nErrorCode := fbMlSvr.nErrorCode;
nMaxInferenceDuration := fbMlSvr.nMaxInferenceDuration;

END_FUNCTION_BLOCK

// ---- POUs/FB_PeriodicLstmSequenceTf3820Runner.TcPOU
FUNCTION_BLOCK FB_PeriodicLstmSequenceTf3820Runner
VAR_INPUT
	sModelJsonFilePath	: T_MaxString;
	sMlSvrNetId			: T_MaxString := 'local';
	eExecutionProvider	: E_ExecutionProvider := E_ExecutionProvider.CPU;
	bEnable				: BOOL;
	bReset					: BOOL;
	bLoadModel			: BOOL;
	nConfigureTimeout	: UDINT := 1000;
	nPredictTimeout		: UDINT := 100;
	nPriority			: UDINT := 0;
	fTheta					: REAL;
	fThetaDot				: REAL;
	fTorque				: REAL;
	fTemperature			: REAL;
	fDirectionFlag		: REAL;
	fThetaStep			: REAL := 0.25;
END_VAR
VAR
	fbMlSvr				: FB_MlSvrPrediction;
	stModelInput		: ST_PeriodicLstmSequenceInput;
	stModelOutput		: ST_PeriodicLstmSequenceOutput;
	rtrig_model			: R_TRIG;
	nState					: INT := 0;
	nSequenceIndex		: INT;
	nOutputIndex		: INT;
END_VAR
VAR_OUTPUT
	bConfigured			: BOOL;
	bBusy					: BOOL;
	bPredictionPending	: BOOL;
	bPredictionReady	: BOOL;
	bResetDone			: BOOL;
	bError					: BOOL;
	nErrorCode			: HRESULT;
	nMaxInferenceDuration	: UDINT;
	aPredictionOutput	: ARRAY[0..8] OF REAL;
END_VAR

rtrig_model(CLK := bLoadModel);

IF rtrig_model.Q THEN
	bPredictionPending := FALSE;
	bPredictionReady := FALSE;
	bResetDone := FALSE;
	bError := FALSE;
	IF fbMlSvr.bConfigured THEN
		nState := 5;
	ELSE
		bConfigured := FALSE;
		nState := 10;
	END_IF
END_IF

IF bReset THEN
	bPredictionPending := FALSE;
	bPredictionReady := FALSE;
	bError := FALSE;
	IF fbMlSvr.bConfigured THEN
		nState := 5;
	ELSE
		bConfigured := FALSE;
		bResetDone := TRUE;
		nState := 0;
	END_IF
END_IF

CASE nState OF
	0:
		bBusy := FALSE;
		IF bLoadModel AND NOT(bConfigured) AND NOT(bReset) THEN
			nState := 10;
		END_IF

	5:
		bBusy := TRUE;
		IF fbMlSvr.Deconfigure(nTimeout := nConfigureTimeout) THEN
			nErrorCode := fbMlSvr.nErrorCode;
			bError := fbMlSvr.bError OR (nErrorCode <> 0);
			bConfigured := FALSE;
			bBusy := FALSE;
			bResetDone := NOT(bError);
			IF bError THEN
				nState := 90;
			ELSIF bReset THEN
				nState := 0;
			ELSE
				nState := 10;
			END_IF
		END_IF

	10:
		bBusy := TRUE;
		fbMlSvr.stPredictionParameter.sMlModelFilePath := sModelJsonFilePath;
		fbMlSvr.stPredictionParameter.sMlSvrNetId := sMlSvrNetId;
		fbMlSvr.stPredictionParameter.eExecutionProvider := eExecutionProvider;
		IF fbMlSvr.Configure(nTimeout := nConfigureTimeout, nPriority := nPriority) THEN
			nErrorCode := fbMlSvr.nErrorCode;
			bError := fbMlSvr.bError OR (nErrorCode <> 0);
			bConfigured := fbMlSvr.bConfigured AND NOT(bError);
			bBusy := FALSE;
			IF bConfigured THEN
				nState := 20;
			ELSE
				nState := 90;
			END_IF
		END_IF

	20:
		bBusy := FALSE;
		bPredictionPending := FALSE;
		IF bEnable AND bConfigured AND NOT(bError) AND NOT(bReset) THEN
			FOR nSequenceIndex := 0 TO 32 DO
				stModelInput.in_input_tensor[0,nSequenceIndex,0] := fTheta + (INT_TO_REAL(nSequenceIndex) * fThetaStep);
				stModelInput.in_input_tensor[0,nSequenceIndex,1] := fThetaDot;
				stModelInput.in_input_tensor[0,nSequenceIndex,2] := fTorque;
				stModelInput.in_input_tensor[0,nSequenceIndex,3] := fTemperature;
				stModelInput.in_input_tensor[0,nSequenceIndex,4] := fDirectionFlag;
			END_FOR
			bPredictionReady := FALSE;
			bPredictionPending := TRUE;
			nState := 30;
		END_IF

	30:
		bBusy := TRUE;
		bPredictionPending := TRUE;
		IF fbMlSvr.Predict(
			pDataIn := ADR(stModelInput),
			nDataInSize := SIZEOF(ST_PeriodicLstmSequenceInput),
			pDataOut := ADR(stModelOutput),
			nDataOutSize := SIZEOF(ST_PeriodicLstmSequenceOutput),
			nTimeout := nPredictTimeout,
			nPriority := nPriority) THEN
			nErrorCode := fbMlSvr.nErrorCode;
			bError := fbMlSvr.bError OR (nErrorCode <> 0);
			nMaxInferenceDuration := fbMlSvr.nMaxInferenceDuration;
			bPredictionPending := FALSE;
			bBusy := FALSE;
			IF NOT(bError) THEN
				aPredictionOutput[0] := stModelOutput.out_prediction_tensor[0,0];
				FOR nOutputIndex := 1 TO 8 DO
					aPredictionOutput[nOutputIndex] := 0.0;
				END_FOR
				bPredictionReady := TRUE;
				nState := 20;
			ELSE
				nState := 90;
			END_IF
		END_IF

	90:
		bBusy := FALSE;
		bPredictionPending := FALSE;
		bError := TRUE;
END_CASE

nErrorCode := fbMlSvr.nErrorCode;
nMaxInferenceDuration := fbMlSvr.nMaxInferenceDuration;

END_FUNCTION_BLOCK

// ---- POUs/FB_PeriodicMlpTf3820Runner.TcPOU
FUNCTION_BLOCK FB_PeriodicMlpTf3820Runner
VAR_INPUT
	sModelJsonFilePath	: T_MaxString;
	sMlSvrNetId			: T_MaxString := 'local';
	eExecutionProvider	: E_ExecutionProvider := E_ExecutionProvider.CPU;
	bEnable				: BOOL;
	bReset					: BOOL;
	bLoadModel			: BOOL;
	nConfigureTimeout	: UDINT := 1000;
	nPredictTimeout		: UDINT := 100;
	nPriority			: UDINT := 0;
	fTheta					: REAL;
	fThetaDot				: REAL;
	fTorque				: REAL;
	fTemperature			: REAL;
	fDirectionFlag		: REAL;
	fThetaStep			: REAL := 0.25;
END_VAR
VAR
	fbMlSvr				: FB_MlSvrPrediction;
	stModelInput		: ST_PeriodicMlpInput;
	stModelOutput		: ST_PeriodicMlpOutput;
	rtrig_model			: R_TRIG;
	nState					: INT := 0;
	nSequenceIndex		: INT;
	nOutputIndex		: INT;
END_VAR
VAR_OUTPUT
	bConfigured			: BOOL;
	bBusy					: BOOL;
	bPredictionPending	: BOOL;
	bPredictionReady	: BOOL;
	bResetDone			: BOOL;
	bError					: BOOL;
	nErrorCode			: HRESULT;
	nMaxInferenceDuration	: UDINT;
	aPredictionOutput	: ARRAY[0..8] OF REAL;
END_VAR

rtrig_model(CLK := bLoadModel);

IF rtrig_model.Q THEN
	bPredictionPending := FALSE;
	bPredictionReady := FALSE;
	bResetDone := FALSE;
	bError := FALSE;
	IF fbMlSvr.bConfigured THEN
		nState := 5;
	ELSE
		bConfigured := FALSE;
		nState := 10;
	END_IF
END_IF

IF bReset THEN
	bPredictionPending := FALSE;
	bPredictionReady := FALSE;
	bError := FALSE;
	IF fbMlSvr.bConfigured THEN
		nState := 5;
	ELSE
		bConfigured := FALSE;
		bResetDone := TRUE;
		nState := 0;
	END_IF
END_IF

CASE nState OF
	0:
		bBusy := FALSE;
		IF bLoadModel AND NOT(bConfigured) AND NOT(bReset) THEN
			nState := 10;
		END_IF

	5:
		bBusy := TRUE;
		IF fbMlSvr.Deconfigure(nTimeout := nConfigureTimeout) THEN
			nErrorCode := fbMlSvr.nErrorCode;
			bError := fbMlSvr.bError OR (nErrorCode <> 0);
			bConfigured := FALSE;
			bBusy := FALSE;
			bResetDone := NOT(bError);
			IF bError THEN
				nState := 90;
			ELSIF bReset THEN
				nState := 0;
			ELSE
				nState := 10;
			END_IF
		END_IF

	10:
		bBusy := TRUE;
		fbMlSvr.stPredictionParameter.sMlModelFilePath := sModelJsonFilePath;
		fbMlSvr.stPredictionParameter.sMlSvrNetId := sMlSvrNetId;
		fbMlSvr.stPredictionParameter.eExecutionProvider := eExecutionProvider;
		IF fbMlSvr.Configure(nTimeout := nConfigureTimeout, nPriority := nPriority) THEN
			nErrorCode := fbMlSvr.nErrorCode;
			bError := fbMlSvr.bError OR (nErrorCode <> 0);
			bConfigured := fbMlSvr.bConfigured AND NOT(bError);
			bBusy := FALSE;
			IF bConfigured THEN
				nState := 20;
			ELSE
				nState := 90;
			END_IF
		END_IF

	20:
		bBusy := FALSE;
		bPredictionPending := FALSE;
		IF bEnable AND bConfigured AND NOT(bError) AND NOT(bReset) THEN
			stModelInput.in_input_tensor[0,0] := fTheta;
			stModelInput.in_input_tensor[0,1] := fThetaDot;
			stModelInput.in_input_tensor[0,2] := fTorque;
			stModelInput.in_input_tensor[0,3] := fTemperature;
			stModelInput.in_input_tensor[0,4] := fDirectionFlag;
			bPredictionReady := FALSE;
			bPredictionPending := TRUE;
			nState := 30;
		END_IF

	30:
		bBusy := TRUE;
		bPredictionPending := TRUE;
		IF fbMlSvr.Predict(
			pDataIn := ADR(stModelInput),
			nDataInSize := SIZEOF(ST_PeriodicMlpInput),
			pDataOut := ADR(stModelOutput),
			nDataOutSize := SIZEOF(ST_PeriodicMlpOutput),
			nTimeout := nPredictTimeout,
			nPriority := nPriority) THEN
			nErrorCode := fbMlSvr.nErrorCode;
			bError := fbMlSvr.bError OR (nErrorCode <> 0);
			nMaxInferenceDuration := fbMlSvr.nMaxInferenceDuration;
			bPredictionPending := FALSE;
			bBusy := FALSE;
			IF NOT(bError) THEN
				aPredictionOutput[0] := stModelOutput.out_prediction_tensor[0,0];
				FOR nOutputIndex := 1 TO 8 DO
					aPredictionOutput[nOutputIndex] := 0.0;
				END_FOR
				bPredictionReady := TRUE;
				nState := 20;
			ELSE
				nState := 90;
			END_IF
		END_IF

	90:
		bBusy := FALSE;
		bPredictionPending := FALSE;
		bError := TRUE;
END_CASE

nErrorCode := fbMlSvr.nErrorCode;
nMaxInferenceDuration := fbMlSvr.nMaxInferenceDuration;

END_FUNCTION_BLOCK

// ---- POUs/FB_PeriodicMlpHarmonicTf3820Runner.TcPOU
FUNCTION_BLOCK FB_PeriodicMlpHarmonicTf3820Runner
VAR_INPUT
	sModelJsonFilePath	: T_MaxString;
	sMlSvrNetId			: T_MaxString := 'local';
	eExecutionProvider	: E_ExecutionProvider := E_ExecutionProvider.CPU;
	bEnable				: BOOL;
	bReset					: BOOL;
	bLoadModel			: BOOL;
	nConfigureTimeout	: UDINT := 1000;
	nPredictTimeout		: UDINT := 100;
	nPriority			: UDINT := 0;
	fTheta					: REAL;
	fThetaDot				: REAL;
	fTorque				: REAL;
	fTemperature			: REAL;
	fDirectionFlag		: REAL;
	fThetaStep			: REAL := 0.25;
END_VAR
VAR
	fbMlSvr				: FB_MlSvrPrediction;
	stModelInput		: ST_PeriodicMlpHarmonicInput;
	stModelOutput		: ST_PeriodicMlpHarmonicOutput;
	rtrig_model			: R_TRIG;
	nState					: INT := 0;
	nSequenceIndex		: INT;
	nOutputIndex		: INT;
END_VAR
VAR_OUTPUT
	bConfigured			: BOOL;
	bBusy					: BOOL;
	bPredictionPending	: BOOL;
	bPredictionReady	: BOOL;
	bResetDone			: BOOL;
	bError					: BOOL;
	nErrorCode			: HRESULT;
	nMaxInferenceDuration	: UDINT;
	aPredictionOutput	: ARRAY[0..8] OF REAL;
END_VAR

rtrig_model(CLK := bLoadModel);

IF rtrig_model.Q THEN
	bPredictionPending := FALSE;
	bPredictionReady := FALSE;
	bResetDone := FALSE;
	bError := FALSE;
	IF fbMlSvr.bConfigured THEN
		nState := 5;
	ELSE
		bConfigured := FALSE;
		nState := 10;
	END_IF
END_IF

IF bReset THEN
	bPredictionPending := FALSE;
	bPredictionReady := FALSE;
	bError := FALSE;
	IF fbMlSvr.bConfigured THEN
		nState := 5;
	ELSE
		bConfigured := FALSE;
		bResetDone := TRUE;
		nState := 0;
	END_IF
END_IF

CASE nState OF
	0:
		bBusy := FALSE;
		IF bLoadModel AND NOT(bConfigured) AND NOT(bReset) THEN
			nState := 10;
		END_IF

	5:
		bBusy := TRUE;
		IF fbMlSvr.Deconfigure(nTimeout := nConfigureTimeout) THEN
			nErrorCode := fbMlSvr.nErrorCode;
			bError := fbMlSvr.bError OR (nErrorCode <> 0);
			bConfigured := FALSE;
			bBusy := FALSE;
			bResetDone := NOT(bError);
			IF bError THEN
				nState := 90;
			ELSIF bReset THEN
				nState := 0;
			ELSE
				nState := 10;
			END_IF
		END_IF

	10:
		bBusy := TRUE;
		fbMlSvr.stPredictionParameter.sMlModelFilePath := sModelJsonFilePath;
		fbMlSvr.stPredictionParameter.sMlSvrNetId := sMlSvrNetId;
		fbMlSvr.stPredictionParameter.eExecutionProvider := eExecutionProvider;
		IF fbMlSvr.Configure(nTimeout := nConfigureTimeout, nPriority := nPriority) THEN
			nErrorCode := fbMlSvr.nErrorCode;
			bError := fbMlSvr.bError OR (nErrorCode <> 0);
			bConfigured := fbMlSvr.bConfigured AND NOT(bError);
			bBusy := FALSE;
			IF bConfigured THEN
				nState := 20;
			ELSE
				nState := 90;
			END_IF
		END_IF

	20:
		bBusy := FALSE;
		bPredictionPending := FALSE;
		IF bEnable AND bConfigured AND NOT(bError) AND NOT(bReset) THEN
			stModelInput.in_input_tensor[0,0] := fTheta;
			stModelInput.in_input_tensor[0,1] := fThetaDot;
			stModelInput.in_input_tensor[0,2] := fTorque;
			stModelInput.in_input_tensor[0,3] := fTemperature;
			stModelInput.in_input_tensor[0,4] := fDirectionFlag;
			bPredictionReady := FALSE;
			bPredictionPending := TRUE;
			nState := 30;
		END_IF

	30:
		bBusy := TRUE;
		bPredictionPending := TRUE;
		IF fbMlSvr.Predict(
			pDataIn := ADR(stModelInput),
			nDataInSize := SIZEOF(ST_PeriodicMlpHarmonicInput),
			pDataOut := ADR(stModelOutput),
			nDataOutSize := SIZEOF(ST_PeriodicMlpHarmonicOutput),
			nTimeout := nPredictTimeout,
			nPriority := nPriority) THEN
			nErrorCode := fbMlSvr.nErrorCode;
			bError := fbMlSvr.bError OR (nErrorCode <> 0);
			nMaxInferenceDuration := fbMlSvr.nMaxInferenceDuration;
			bPredictionPending := FALSE;
			bBusy := FALSE;
			IF NOT(bError) THEN
				aPredictionOutput[0] := stModelOutput.out_prediction_tensor[0,0];
				FOR nOutputIndex := 1 TO 8 DO
					aPredictionOutput[nOutputIndex] := 0.0;
				END_FOR
				bPredictionReady := TRUE;
				nState := 20;
			ELSE
				nState := 90;
			END_IF
		END_IF

	90:
		bBusy := FALSE;
		bPredictionPending := FALSE;
		bError := TRUE;
END_CASE

nErrorCode := fbMlSvr.nErrorCode;
nMaxInferenceDuration := fbMlSvr.nMaxInferenceDuration;

END_FUNCTION_BLOCK

// ---- POUs/FB_PeriodicTemporalConvolutionTf3820Runner.TcPOU
FUNCTION_BLOCK FB_PeriodicTemporalConvolutionTf3820Runner
VAR_INPUT
	sModelJsonFilePath	: T_MaxString;
	sMlSvrNetId			: T_MaxString := 'local';
	eExecutionProvider	: E_ExecutionProvider := E_ExecutionProvider.CPU;
	bEnable				: BOOL;
	bReset					: BOOL;
	bLoadModel			: BOOL;
	nConfigureTimeout	: UDINT := 1000;
	nPredictTimeout		: UDINT := 100;
	nPriority			: UDINT := 0;
	fTheta					: REAL;
	fThetaDot				: REAL;
	fTorque				: REAL;
	fTemperature			: REAL;
	fDirectionFlag		: REAL;
	fThetaStep			: REAL := 0.25;
END_VAR
VAR
	fbMlSvr				: FB_MlSvrPrediction;
	stModelInput		: ST_PeriodicTemporalConvolutionInput;
	stModelOutput		: ST_PeriodicTemporalConvolutionOutput;
	rtrig_model			: R_TRIG;
	nState					: INT := 0;
	nSequenceIndex		: INT;
	nOutputIndex		: INT;
END_VAR
VAR_OUTPUT
	bConfigured			: BOOL;
	bBusy					: BOOL;
	bPredictionPending	: BOOL;
	bPredictionReady	: BOOL;
	bResetDone			: BOOL;
	bError					: BOOL;
	nErrorCode			: HRESULT;
	nMaxInferenceDuration	: UDINT;
	aPredictionOutput	: ARRAY[0..8] OF REAL;
END_VAR

rtrig_model(CLK := bLoadModel);

IF rtrig_model.Q THEN
	bPredictionPending := FALSE;
	bPredictionReady := FALSE;
	bResetDone := FALSE;
	bError := FALSE;
	IF fbMlSvr.bConfigured THEN
		nState := 5;
	ELSE
		bConfigured := FALSE;
		nState := 10;
	END_IF
END_IF

IF bReset THEN
	bPredictionPending := FALSE;
	bPredictionReady := FALSE;
	bError := FALSE;
	IF fbMlSvr.bConfigured THEN
		nState := 5;
	ELSE
		bConfigured := FALSE;
		bResetDone := TRUE;
		nState := 0;
	END_IF
END_IF

CASE nState OF
	0:
		bBusy := FALSE;
		IF bLoadModel AND NOT(bConfigured) AND NOT(bReset) THEN
			nState := 10;
		END_IF

	5:
		bBusy := TRUE;
		IF fbMlSvr.Deconfigure(nTimeout := nConfigureTimeout) THEN
			nErrorCode := fbMlSvr.nErrorCode;
			bError := fbMlSvr.bError OR (nErrorCode <> 0);
			bConfigured := FALSE;
			bBusy := FALSE;
			bResetDone := NOT(bError);
			IF bError THEN
				nState := 90;
			ELSIF bReset THEN
				nState := 0;
			ELSE
				nState := 10;
			END_IF
		END_IF

	10:
		bBusy := TRUE;
		fbMlSvr.stPredictionParameter.sMlModelFilePath := sModelJsonFilePath;
		fbMlSvr.stPredictionParameter.sMlSvrNetId := sMlSvrNetId;
		fbMlSvr.stPredictionParameter.eExecutionProvider := eExecutionProvider;
		IF fbMlSvr.Configure(nTimeout := nConfigureTimeout, nPriority := nPriority) THEN
			nErrorCode := fbMlSvr.nErrorCode;
			bError := fbMlSvr.bError OR (nErrorCode <> 0);
			bConfigured := fbMlSvr.bConfigured AND NOT(bError);
			bBusy := FALSE;
			IF bConfigured THEN
				nState := 20;
			ELSE
				nState := 90;
			END_IF
		END_IF

	20:
		bBusy := FALSE;
		bPredictionPending := FALSE;
		IF bEnable AND bConfigured AND NOT(bError) AND NOT(bReset) THEN
			FOR nSequenceIndex := 0 TO 32 DO
				stModelInput.in_input_tensor[0,nSequenceIndex,0] := fTheta + (INT_TO_REAL(nSequenceIndex) * fThetaStep);
				stModelInput.in_input_tensor[0,nSequenceIndex,1] := fThetaDot;
				stModelInput.in_input_tensor[0,nSequenceIndex,2] := fTorque;
				stModelInput.in_input_tensor[0,nSequenceIndex,3] := fTemperature;
				stModelInput.in_input_tensor[0,nSequenceIndex,4] := fDirectionFlag;
			END_FOR
			bPredictionReady := FALSE;
			bPredictionPending := TRUE;
			nState := 30;
		END_IF

	30:
		bBusy := TRUE;
		bPredictionPending := TRUE;
		IF fbMlSvr.Predict(
			pDataIn := ADR(stModelInput),
			nDataInSize := SIZEOF(ST_PeriodicTemporalConvolutionInput),
			pDataOut := ADR(stModelOutput),
			nDataOutSize := SIZEOF(ST_PeriodicTemporalConvolutionOutput),
			nTimeout := nPredictTimeout,
			nPriority := nPriority) THEN
			nErrorCode := fbMlSvr.nErrorCode;
			bError := fbMlSvr.bError OR (nErrorCode <> 0);
			nMaxInferenceDuration := fbMlSvr.nMaxInferenceDuration;
			bPredictionPending := FALSE;
			bBusy := FALSE;
			IF NOT(bError) THEN
				aPredictionOutput[0] := stModelOutput.out_prediction_tensor[0,0];
				FOR nOutputIndex := 1 TO 8 DO
					aPredictionOutput[nOutputIndex] := 0.0;
				END_FOR
				bPredictionReady := TRUE;
				nState := 20;
			ELSE
				nState := 90;
			END_IF
		END_IF

	90:
		bBusy := FALSE;
		bPredictionPending := FALSE;
		bError := TRUE;
END_CASE

nErrorCode := fbMlSvr.nErrorCode;
nMaxInferenceDuration := fbMlSvr.nMaxInferenceDuration;

END_FUNCTION_BLOCK

// ---- POUs/FB_RcimTrack1Tf3820Runner.TcPOU
FUNCTION_BLOCK FB_RcimTrack1Tf3820Runner
VAR_INPUT
	sModelJsonFilePath	: T_MaxString;
	sMlSvrNetId			: T_MaxString := 'local';
	eExecutionProvider	: E_ExecutionProvider := E_ExecutionProvider.CPU;
	bEnable				: BOOL;
	bReset					: BOOL;
	bLoadModel			: BOOL;
	nConfigureTimeout	: UDINT := 1000;
	nPredictTimeout		: UDINT := 100;
	nPriority			: UDINT := 0;
	fTheta					: REAL;
	fThetaDot				: REAL;
	fTorque				: REAL;
	fTemperature			: REAL;
	fDirectionFlag		: REAL;
	fThetaStep			: REAL := 0.25;
END_VAR
VAR
	fbMlSvr				: FB_MlSvrPrediction;
	stModelInput		: ST_RcimTrack1Input;
	stModelOutput		: ST_RcimTrack1Output;
	rtrig_model			: R_TRIG;
	nState					: INT := 0;
	nSequenceIndex		: INT;
	nOutputIndex		: INT;
END_VAR
VAR_OUTPUT
	bConfigured			: BOOL;
	bBusy					: BOOL;
	bPredictionPending	: BOOL;
	bPredictionReady	: BOOL;
	bResetDone			: BOOL;
	bError					: BOOL;
	nErrorCode			: HRESULT;
	nMaxInferenceDuration	: UDINT;
	aPredictionOutput	: ARRAY[0..8] OF REAL;
END_VAR

rtrig_model(CLK := bLoadModel);

IF rtrig_model.Q THEN
	bPredictionPending := FALSE;
	bPredictionReady := FALSE;
	bResetDone := FALSE;
	bError := FALSE;
	IF fbMlSvr.bConfigured THEN
		nState := 5;
	ELSE
		bConfigured := FALSE;
		nState := 10;
	END_IF
END_IF

IF bReset THEN
	bPredictionPending := FALSE;
	bPredictionReady := FALSE;
	bError := FALSE;
	IF fbMlSvr.bConfigured THEN
		nState := 5;
	ELSE
		bConfigured := FALSE;
		bResetDone := TRUE;
		nState := 0;
	END_IF
END_IF

CASE nState OF
	0:
		bBusy := FALSE;
		IF bLoadModel AND NOT(bConfigured) AND NOT(bReset) THEN
			nState := 10;
		END_IF

	5:
		bBusy := TRUE;
		IF fbMlSvr.Deconfigure(nTimeout := nConfigureTimeout) THEN
			nErrorCode := fbMlSvr.nErrorCode;
			bError := fbMlSvr.bError OR (nErrorCode <> 0);
			bConfigured := FALSE;
			bBusy := FALSE;
			bResetDone := NOT(bError);
			IF bError THEN
				nState := 90;
			ELSIF bReset THEN
				nState := 0;
			ELSE
				nState := 10;
			END_IF
		END_IF

	10:
		bBusy := TRUE;
		fbMlSvr.stPredictionParameter.sMlModelFilePath := sModelJsonFilePath;
		fbMlSvr.stPredictionParameter.sMlSvrNetId := sMlSvrNetId;
		fbMlSvr.stPredictionParameter.eExecutionProvider := eExecutionProvider;
		IF fbMlSvr.Configure(nTimeout := nConfigureTimeout, nPriority := nPriority) THEN
			nErrorCode := fbMlSvr.nErrorCode;
			bError := fbMlSvr.bError OR (nErrorCode <> 0);
			bConfigured := fbMlSvr.bConfigured AND NOT(bError);
			bBusy := FALSE;
			IF bConfigured THEN
				nState := 20;
			ELSE
				nState := 90;
			END_IF
		END_IF

	20:
		bBusy := FALSE;
		bPredictionPending := FALSE;
		IF bEnable AND bConfigured AND NOT(bError) AND NOT(bReset) THEN
			stModelInput.in_float_input[0,0] := fThetaDot;
			stModelInput.in_float_input[0,1] := fTemperature;
			stModelInput.in_float_input[0,2] := fTorque;
			bPredictionReady := FALSE;
			bPredictionPending := TRUE;
			nState := 30;
		END_IF

	30:
		bBusy := TRUE;
		bPredictionPending := TRUE;
		IF fbMlSvr.Predict(
			pDataIn := ADR(stModelInput),
			nDataInSize := SIZEOF(ST_RcimTrack1Input),
			pDataOut := ADR(stModelOutput),
			nDataOutSize := SIZEOF(ST_RcimTrack1Output),
			nTimeout := nPredictTimeout,
			nPriority := nPriority) THEN
			nErrorCode := fbMlSvr.nErrorCode;
			bError := fbMlSvr.bError OR (nErrorCode <> 0);
			nMaxInferenceDuration := fbMlSvr.nMaxInferenceDuration;
			bPredictionPending := FALSE;
			bBusy := FALSE;
			IF NOT(bError) THEN
				aPredictionOutput[0] := stModelOutput.out_variable[0,0];
				FOR nOutputIndex := 1 TO 8 DO
					aPredictionOutput[nOutputIndex] := 0.0;
				END_FOR
				bPredictionReady := TRUE;
				nState := 20;
			ELSE
				nState := 90;
			END_IF
		END_IF

	90:
		bBusy := FALSE;
		bPredictionPending := FALSE;
		bError := TRUE;
END_CASE

nErrorCode := fbMlSvr.nErrorCode;
nMaxInferenceDuration := fbMlSvr.nMaxInferenceDuration;

END_FUNCTION_BLOCK

// ---- POUs/FB_ResidualHarmonicGruSequenceDense240Tf3820Runner.TcPOU
FUNCTION_BLOCK FB_ResidualHarmonicGruSequenceDense240Tf3820Runner
VAR_INPUT
	sModelJsonFilePath	: T_MaxString;
	sMlSvrNetId			: T_MaxString := 'local';
	eExecutionProvider	: E_ExecutionProvider := E_ExecutionProvider.CPU;
	bEnable				: BOOL;
	bReset					: BOOL;
	bLoadModel			: BOOL;
	nConfigureTimeout	: UDINT := 1000;
	nPredictTimeout		: UDINT := 100;
	nPriority			: UDINT := 0;
	fTheta					: REAL;
	fThetaDot				: REAL;
	fTorque				: REAL;
	fTemperature			: REAL;
	fDirectionFlag		: REAL;
	fThetaStep			: REAL := 0.25;
END_VAR
VAR
	fbMlSvr				: FB_MlSvrPrediction;
	stModelInput		: ST_ResidualHarmonicGruSequenceDense240Input;
	stModelOutput		: ST_ResidualHarmonicGruSequenceDense240Output;
	rtrig_model			: R_TRIG;
	nState					: INT := 0;
	nSequenceIndex		: INT;
	nOutputIndex		: INT;
END_VAR
VAR_OUTPUT
	bConfigured			: BOOL;
	bBusy					: BOOL;
	bPredictionPending	: BOOL;
	bPredictionReady	: BOOL;
	bResetDone			: BOOL;
	bError					: BOOL;
	nErrorCode			: HRESULT;
	nMaxInferenceDuration	: UDINT;
	aPredictionOutput	: ARRAY[0..8] OF REAL;
END_VAR

rtrig_model(CLK := bLoadModel);

IF rtrig_model.Q THEN
	bPredictionPending := FALSE;
	bPredictionReady := FALSE;
	bResetDone := FALSE;
	bError := FALSE;
	IF fbMlSvr.bConfigured THEN
		nState := 5;
	ELSE
		bConfigured := FALSE;
		nState := 10;
	END_IF
END_IF

IF bReset THEN
	bPredictionPending := FALSE;
	bPredictionReady := FALSE;
	bError := FALSE;
	IF fbMlSvr.bConfigured THEN
		nState := 5;
	ELSE
		bConfigured := FALSE;
		bResetDone := TRUE;
		nState := 0;
	END_IF
END_IF

CASE nState OF
	0:
		bBusy := FALSE;
		IF bLoadModel AND NOT(bConfigured) AND NOT(bReset) THEN
			nState := 10;
		END_IF

	5:
		bBusy := TRUE;
		IF fbMlSvr.Deconfigure(nTimeout := nConfigureTimeout) THEN
			nErrorCode := fbMlSvr.nErrorCode;
			bError := fbMlSvr.bError OR (nErrorCode <> 0);
			bConfigured := FALSE;
			bBusy := FALSE;
			bResetDone := NOT(bError);
			IF bError THEN
				nState := 90;
			ELSIF bReset THEN
				nState := 0;
			ELSE
				nState := 10;
			END_IF
		END_IF

	10:
		bBusy := TRUE;
		fbMlSvr.stPredictionParameter.sMlModelFilePath := sModelJsonFilePath;
		fbMlSvr.stPredictionParameter.sMlSvrNetId := sMlSvrNetId;
		fbMlSvr.stPredictionParameter.eExecutionProvider := eExecutionProvider;
		IF fbMlSvr.Configure(nTimeout := nConfigureTimeout, nPriority := nPriority) THEN
			nErrorCode := fbMlSvr.nErrorCode;
			bError := fbMlSvr.bError OR (nErrorCode <> 0);
			bConfigured := fbMlSvr.bConfigured AND NOT(bError);
			bBusy := FALSE;
			IF bConfigured THEN
				nState := 20;
			ELSE
				nState := 90;
			END_IF
		END_IF

	20:
		bBusy := FALSE;
		bPredictionPending := FALSE;
		IF bEnable AND bConfigured AND NOT(bError) AND NOT(bReset) THEN
			FOR nSequenceIndex := 0 TO 32 DO
				stModelInput.in_input_tensor[0,nSequenceIndex,0] := fTheta + (INT_TO_REAL(nSequenceIndex) * fThetaStep);
				stModelInput.in_input_tensor[0,nSequenceIndex,1] := fThetaDot;
				stModelInput.in_input_tensor[0,nSequenceIndex,2] := fTorque;
				stModelInput.in_input_tensor[0,nSequenceIndex,3] := fTemperature;
				stModelInput.in_input_tensor[0,nSequenceIndex,4] := fDirectionFlag;
			END_FOR
			bPredictionReady := FALSE;
			bPredictionPending := TRUE;
			nState := 30;
		END_IF

	30:
		bBusy := TRUE;
		bPredictionPending := TRUE;
		IF fbMlSvr.Predict(
			pDataIn := ADR(stModelInput),
			nDataInSize := SIZEOF(ST_ResidualHarmonicGruSequenceDense240Input),
			pDataOut := ADR(stModelOutput),
			nDataOutSize := SIZEOF(ST_ResidualHarmonicGruSequenceDense240Output),
			nTimeout := nPredictTimeout,
			nPriority := nPriority) THEN
			nErrorCode := fbMlSvr.nErrorCode;
			bError := fbMlSvr.bError OR (nErrorCode <> 0);
			nMaxInferenceDuration := fbMlSvr.nMaxInferenceDuration;
			bPredictionPending := FALSE;
			bBusy := FALSE;
			IF NOT(bError) THEN
				aPredictionOutput[0] := stModelOutput.out_prediction_tensor[0,0];
				FOR nOutputIndex := 1 TO 8 DO
					aPredictionOutput[nOutputIndex] := 0.0;
				END_FOR
				bPredictionReady := TRUE;
				nState := 20;
			ELSE
				nState := 90;
			END_IF
		END_IF

	90:
		bBusy := FALSE;
		bPredictionPending := FALSE;
		bError := TRUE;
END_CASE

nErrorCode := fbMlSvr.nErrorCode;
nMaxInferenceDuration := fbMlSvr.nMaxInferenceDuration;

END_FUNCTION_BLOCK

// ---- POUs/FB_ResidualHarmonicGruSequenceDense360Tf3820Runner.TcPOU
FUNCTION_BLOCK FB_ResidualHarmonicGruSequenceDense360Tf3820Runner
VAR_INPUT
	sModelJsonFilePath	: T_MaxString;
	sMlSvrNetId			: T_MaxString := 'local';
	eExecutionProvider	: E_ExecutionProvider := E_ExecutionProvider.CPU;
	bEnable				: BOOL;
	bReset					: BOOL;
	bLoadModel			: BOOL;
	nConfigureTimeout	: UDINT := 1000;
	nPredictTimeout		: UDINT := 100;
	nPriority			: UDINT := 0;
	fTheta					: REAL;
	fThetaDot				: REAL;
	fTorque				: REAL;
	fTemperature			: REAL;
	fDirectionFlag		: REAL;
	fThetaStep			: REAL := 0.25;
END_VAR
VAR
	fbMlSvr				: FB_MlSvrPrediction;
	stModelInput		: ST_ResidualHarmonicGruSequenceDense360Input;
	stModelOutput		: ST_ResidualHarmonicGruSequenceDense360Output;
	rtrig_model			: R_TRIG;
	nState					: INT := 0;
	nSequenceIndex		: INT;
	nOutputIndex		: INT;
END_VAR
VAR_OUTPUT
	bConfigured			: BOOL;
	bBusy					: BOOL;
	bPredictionPending	: BOOL;
	bPredictionReady	: BOOL;
	bResetDone			: BOOL;
	bError					: BOOL;
	nErrorCode			: HRESULT;
	nMaxInferenceDuration	: UDINT;
	aPredictionOutput	: ARRAY[0..8] OF REAL;
END_VAR

rtrig_model(CLK := bLoadModel);

IF rtrig_model.Q THEN
	bPredictionPending := FALSE;
	bPredictionReady := FALSE;
	bResetDone := FALSE;
	bError := FALSE;
	IF fbMlSvr.bConfigured THEN
		nState := 5;
	ELSE
		bConfigured := FALSE;
		nState := 10;
	END_IF
END_IF

IF bReset THEN
	bPredictionPending := FALSE;
	bPredictionReady := FALSE;
	bError := FALSE;
	IF fbMlSvr.bConfigured THEN
		nState := 5;
	ELSE
		bConfigured := FALSE;
		bResetDone := TRUE;
		nState := 0;
	END_IF
END_IF

CASE nState OF
	0:
		bBusy := FALSE;
		IF bLoadModel AND NOT(bConfigured) AND NOT(bReset) THEN
			nState := 10;
		END_IF

	5:
		bBusy := TRUE;
		IF fbMlSvr.Deconfigure(nTimeout := nConfigureTimeout) THEN
			nErrorCode := fbMlSvr.nErrorCode;
			bError := fbMlSvr.bError OR (nErrorCode <> 0);
			bConfigured := FALSE;
			bBusy := FALSE;
			bResetDone := NOT(bError);
			IF bError THEN
				nState := 90;
			ELSIF bReset THEN
				nState := 0;
			ELSE
				nState := 10;
			END_IF
		END_IF

	10:
		bBusy := TRUE;
		fbMlSvr.stPredictionParameter.sMlModelFilePath := sModelJsonFilePath;
		fbMlSvr.stPredictionParameter.sMlSvrNetId := sMlSvrNetId;
		fbMlSvr.stPredictionParameter.eExecutionProvider := eExecutionProvider;
		IF fbMlSvr.Configure(nTimeout := nConfigureTimeout, nPriority := nPriority) THEN
			nErrorCode := fbMlSvr.nErrorCode;
			bError := fbMlSvr.bError OR (nErrorCode <> 0);
			bConfigured := fbMlSvr.bConfigured AND NOT(bError);
			bBusy := FALSE;
			IF bConfigured THEN
				nState := 20;
			ELSE
				nState := 90;
			END_IF
		END_IF

	20:
		bBusy := FALSE;
		bPredictionPending := FALSE;
		IF bEnable AND bConfigured AND NOT(bError) AND NOT(bReset) THEN
			FOR nSequenceIndex := 0 TO 32 DO
				stModelInput.in_input_tensor[0,nSequenceIndex,0] := fTheta + (INT_TO_REAL(nSequenceIndex) * fThetaStep);
				stModelInput.in_input_tensor[0,nSequenceIndex,1] := fThetaDot;
				stModelInput.in_input_tensor[0,nSequenceIndex,2] := fTorque;
				stModelInput.in_input_tensor[0,nSequenceIndex,3] := fTemperature;
				stModelInput.in_input_tensor[0,nSequenceIndex,4] := fDirectionFlag;
			END_FOR
			bPredictionReady := FALSE;
			bPredictionPending := TRUE;
			nState := 30;
		END_IF

	30:
		bBusy := TRUE;
		bPredictionPending := TRUE;
		IF fbMlSvr.Predict(
			pDataIn := ADR(stModelInput),
			nDataInSize := SIZEOF(ST_ResidualHarmonicGruSequenceDense360Input),
			pDataOut := ADR(stModelOutput),
			nDataOutSize := SIZEOF(ST_ResidualHarmonicGruSequenceDense360Output),
			nTimeout := nPredictTimeout,
			nPriority := nPriority) THEN
			nErrorCode := fbMlSvr.nErrorCode;
			bError := fbMlSvr.bError OR (nErrorCode <> 0);
			nMaxInferenceDuration := fbMlSvr.nMaxInferenceDuration;
			bPredictionPending := FALSE;
			bBusy := FALSE;
			IF NOT(bError) THEN
				aPredictionOutput[0] := stModelOutput.out_prediction_tensor[0,0];
				FOR nOutputIndex := 1 TO 8 DO
					aPredictionOutput[nOutputIndex] := 0.0;
				END_FOR
				bPredictionReady := TRUE;
				nState := 20;
			ELSE
				nState := 90;
			END_IF
		END_IF

	90:
		bBusy := FALSE;
		bPredictionPending := FALSE;
		bError := TRUE;
END_CASE

nErrorCode := fbMlSvr.nErrorCode;
nMaxInferenceDuration := fbMlSvr.nMaxInferenceDuration;

END_FUNCTION_BLOCK

// ---- POUs/FB_ResidualHarmonicGruSequenceSparseRcimTf3820Runner.TcPOU
FUNCTION_BLOCK FB_ResidualHarmonicGruSequenceSparseRcimTf3820Runner
VAR_INPUT
	sModelJsonFilePath	: T_MaxString;
	sMlSvrNetId			: T_MaxString := 'local';
	eExecutionProvider	: E_ExecutionProvider := E_ExecutionProvider.CPU;
	bEnable				: BOOL;
	bReset					: BOOL;
	bLoadModel			: BOOL;
	nConfigureTimeout	: UDINT := 1000;
	nPredictTimeout		: UDINT := 100;
	nPriority			: UDINT := 0;
	fTheta					: REAL;
	fThetaDot				: REAL;
	fTorque				: REAL;
	fTemperature			: REAL;
	fDirectionFlag		: REAL;
	fThetaStep			: REAL := 0.25;
END_VAR
VAR
	fbMlSvr				: FB_MlSvrPrediction;
	stModelInput		: ST_ResidualHarmonicGruSequenceSparseRcimInput;
	stModelOutput		: ST_ResidualHarmonicGruSequenceSparseRcimOutput;
	rtrig_model			: R_TRIG;
	nState					: INT := 0;
	nSequenceIndex		: INT;
	nOutputIndex		: INT;
END_VAR
VAR_OUTPUT
	bConfigured			: BOOL;
	bBusy					: BOOL;
	bPredictionPending	: BOOL;
	bPredictionReady	: BOOL;
	bResetDone			: BOOL;
	bError					: BOOL;
	nErrorCode			: HRESULT;
	nMaxInferenceDuration	: UDINT;
	aPredictionOutput	: ARRAY[0..8] OF REAL;
END_VAR

rtrig_model(CLK := bLoadModel);

IF rtrig_model.Q THEN
	bPredictionPending := FALSE;
	bPredictionReady := FALSE;
	bResetDone := FALSE;
	bError := FALSE;
	IF fbMlSvr.bConfigured THEN
		nState := 5;
	ELSE
		bConfigured := FALSE;
		nState := 10;
	END_IF
END_IF

IF bReset THEN
	bPredictionPending := FALSE;
	bPredictionReady := FALSE;
	bError := FALSE;
	IF fbMlSvr.bConfigured THEN
		nState := 5;
	ELSE
		bConfigured := FALSE;
		bResetDone := TRUE;
		nState := 0;
	END_IF
END_IF

CASE nState OF
	0:
		bBusy := FALSE;
		IF bLoadModel AND NOT(bConfigured) AND NOT(bReset) THEN
			nState := 10;
		END_IF

	5:
		bBusy := TRUE;
		IF fbMlSvr.Deconfigure(nTimeout := nConfigureTimeout) THEN
			nErrorCode := fbMlSvr.nErrorCode;
			bError := fbMlSvr.bError OR (nErrorCode <> 0);
			bConfigured := FALSE;
			bBusy := FALSE;
			bResetDone := NOT(bError);
			IF bError THEN
				nState := 90;
			ELSIF bReset THEN
				nState := 0;
			ELSE
				nState := 10;
			END_IF
		END_IF

	10:
		bBusy := TRUE;
		fbMlSvr.stPredictionParameter.sMlModelFilePath := sModelJsonFilePath;
		fbMlSvr.stPredictionParameter.sMlSvrNetId := sMlSvrNetId;
		fbMlSvr.stPredictionParameter.eExecutionProvider := eExecutionProvider;
		IF fbMlSvr.Configure(nTimeout := nConfigureTimeout, nPriority := nPriority) THEN
			nErrorCode := fbMlSvr.nErrorCode;
			bError := fbMlSvr.bError OR (nErrorCode <> 0);
			bConfigured := fbMlSvr.bConfigured AND NOT(bError);
			bBusy := FALSE;
			IF bConfigured THEN
				nState := 20;
			ELSE
				nState := 90;
			END_IF
		END_IF

	20:
		bBusy := FALSE;
		bPredictionPending := FALSE;
		IF bEnable AND bConfigured AND NOT(bError) AND NOT(bReset) THEN
			FOR nSequenceIndex := 0 TO 32 DO
				stModelInput.in_input_tensor[0,nSequenceIndex,0] := fTheta + (INT_TO_REAL(nSequenceIndex) * fThetaStep);
				stModelInput.in_input_tensor[0,nSequenceIndex,1] := fThetaDot;
				stModelInput.in_input_tensor[0,nSequenceIndex,2] := fTorque;
				stModelInput.in_input_tensor[0,nSequenceIndex,3] := fTemperature;
				stModelInput.in_input_tensor[0,nSequenceIndex,4] := fDirectionFlag;
			END_FOR
			bPredictionReady := FALSE;
			bPredictionPending := TRUE;
			nState := 30;
		END_IF

	30:
		bBusy := TRUE;
		bPredictionPending := TRUE;
		IF fbMlSvr.Predict(
			pDataIn := ADR(stModelInput),
			nDataInSize := SIZEOF(ST_ResidualHarmonicGruSequenceSparseRcimInput),
			pDataOut := ADR(stModelOutput),
			nDataOutSize := SIZEOF(ST_ResidualHarmonicGruSequenceSparseRcimOutput),
			nTimeout := nPredictTimeout,
			nPriority := nPriority) THEN
			nErrorCode := fbMlSvr.nErrorCode;
			bError := fbMlSvr.bError OR (nErrorCode <> 0);
			nMaxInferenceDuration := fbMlSvr.nMaxInferenceDuration;
			bPredictionPending := FALSE;
			bBusy := FALSE;
			IF NOT(bError) THEN
				aPredictionOutput[0] := stModelOutput.out_prediction_tensor[0,0];
				FOR nOutputIndex := 1 TO 8 DO
					aPredictionOutput[nOutputIndex] := 0.0;
				END_FOR
				bPredictionReady := TRUE;
				nState := 20;
			ELSE
				nState := 90;
			END_IF
		END_IF

	90:
		bBusy := FALSE;
		bPredictionPending := FALSE;
		bError := TRUE;
END_CASE

nErrorCode := fbMlSvr.nErrorCode;
nMaxInferenceDuration := fbMlSvr.nMaxInferenceDuration;

END_FUNCTION_BLOCK

// ---- POUs/FB_ResidualHarmonicLstmSequenceDense240Tf3820Runner.TcPOU
FUNCTION_BLOCK FB_ResidualHarmonicLstmSequenceDense240Tf3820Runner
VAR_INPUT
	sModelJsonFilePath	: T_MaxString;
	sMlSvrNetId			: T_MaxString := 'local';
	eExecutionProvider	: E_ExecutionProvider := E_ExecutionProvider.CPU;
	bEnable				: BOOL;
	bReset					: BOOL;
	bLoadModel			: BOOL;
	nConfigureTimeout	: UDINT := 1000;
	nPredictTimeout		: UDINT := 100;
	nPriority			: UDINT := 0;
	fTheta					: REAL;
	fThetaDot				: REAL;
	fTorque				: REAL;
	fTemperature			: REAL;
	fDirectionFlag		: REAL;
	fThetaStep			: REAL := 0.25;
END_VAR
VAR
	fbMlSvr				: FB_MlSvrPrediction;
	stModelInput		: ST_ResidualHarmonicLstmSequenceDense240Input;
	stModelOutput		: ST_ResidualHarmonicLstmSequenceDense240Output;
	rtrig_model			: R_TRIG;
	nState					: INT := 0;
	nSequenceIndex		: INT;
	nOutputIndex		: INT;
END_VAR
VAR_OUTPUT
	bConfigured			: BOOL;
	bBusy					: BOOL;
	bPredictionPending	: BOOL;
	bPredictionReady	: BOOL;
	bResetDone			: BOOL;
	bError					: BOOL;
	nErrorCode			: HRESULT;
	nMaxInferenceDuration	: UDINT;
	aPredictionOutput	: ARRAY[0..8] OF REAL;
END_VAR

rtrig_model(CLK := bLoadModel);

IF rtrig_model.Q THEN
	bPredictionPending := FALSE;
	bPredictionReady := FALSE;
	bResetDone := FALSE;
	bError := FALSE;
	IF fbMlSvr.bConfigured THEN
		nState := 5;
	ELSE
		bConfigured := FALSE;
		nState := 10;
	END_IF
END_IF

IF bReset THEN
	bPredictionPending := FALSE;
	bPredictionReady := FALSE;
	bError := FALSE;
	IF fbMlSvr.bConfigured THEN
		nState := 5;
	ELSE
		bConfigured := FALSE;
		bResetDone := TRUE;
		nState := 0;
	END_IF
END_IF

CASE nState OF
	0:
		bBusy := FALSE;
		IF bLoadModel AND NOT(bConfigured) AND NOT(bReset) THEN
			nState := 10;
		END_IF

	5:
		bBusy := TRUE;
		IF fbMlSvr.Deconfigure(nTimeout := nConfigureTimeout) THEN
			nErrorCode := fbMlSvr.nErrorCode;
			bError := fbMlSvr.bError OR (nErrorCode <> 0);
			bConfigured := FALSE;
			bBusy := FALSE;
			bResetDone := NOT(bError);
			IF bError THEN
				nState := 90;
			ELSIF bReset THEN
				nState := 0;
			ELSE
				nState := 10;
			END_IF
		END_IF

	10:
		bBusy := TRUE;
		fbMlSvr.stPredictionParameter.sMlModelFilePath := sModelJsonFilePath;
		fbMlSvr.stPredictionParameter.sMlSvrNetId := sMlSvrNetId;
		fbMlSvr.stPredictionParameter.eExecutionProvider := eExecutionProvider;
		IF fbMlSvr.Configure(nTimeout := nConfigureTimeout, nPriority := nPriority) THEN
			nErrorCode := fbMlSvr.nErrorCode;
			bError := fbMlSvr.bError OR (nErrorCode <> 0);
			bConfigured := fbMlSvr.bConfigured AND NOT(bError);
			bBusy := FALSE;
			IF bConfigured THEN
				nState := 20;
			ELSE
				nState := 90;
			END_IF
		END_IF

	20:
		bBusy := FALSE;
		bPredictionPending := FALSE;
		IF bEnable AND bConfigured AND NOT(bError) AND NOT(bReset) THEN
			FOR nSequenceIndex := 0 TO 32 DO
				stModelInput.in_input_tensor[0,nSequenceIndex,0] := fTheta + (INT_TO_REAL(nSequenceIndex) * fThetaStep);
				stModelInput.in_input_tensor[0,nSequenceIndex,1] := fThetaDot;
				stModelInput.in_input_tensor[0,nSequenceIndex,2] := fTorque;
				stModelInput.in_input_tensor[0,nSequenceIndex,3] := fTemperature;
				stModelInput.in_input_tensor[0,nSequenceIndex,4] := fDirectionFlag;
			END_FOR
			bPredictionReady := FALSE;
			bPredictionPending := TRUE;
			nState := 30;
		END_IF

	30:
		bBusy := TRUE;
		bPredictionPending := TRUE;
		IF fbMlSvr.Predict(
			pDataIn := ADR(stModelInput),
			nDataInSize := SIZEOF(ST_ResidualHarmonicLstmSequenceDense240Input),
			pDataOut := ADR(stModelOutput),
			nDataOutSize := SIZEOF(ST_ResidualHarmonicLstmSequenceDense240Output),
			nTimeout := nPredictTimeout,
			nPriority := nPriority) THEN
			nErrorCode := fbMlSvr.nErrorCode;
			bError := fbMlSvr.bError OR (nErrorCode <> 0);
			nMaxInferenceDuration := fbMlSvr.nMaxInferenceDuration;
			bPredictionPending := FALSE;
			bBusy := FALSE;
			IF NOT(bError) THEN
				aPredictionOutput[0] := stModelOutput.out_prediction_tensor[0,0];
				FOR nOutputIndex := 1 TO 8 DO
					aPredictionOutput[nOutputIndex] := 0.0;
				END_FOR
				bPredictionReady := TRUE;
				nState := 20;
			ELSE
				nState := 90;
			END_IF
		END_IF

	90:
		bBusy := FALSE;
		bPredictionPending := FALSE;
		bError := TRUE;
END_CASE

nErrorCode := fbMlSvr.nErrorCode;
nMaxInferenceDuration := fbMlSvr.nMaxInferenceDuration;

END_FUNCTION_BLOCK

// ---- POUs/FB_ResidualHarmonicLstmSequenceDense360Tf3820Runner.TcPOU
FUNCTION_BLOCK FB_ResidualHarmonicLstmSequenceDense360Tf3820Runner
VAR_INPUT
	sModelJsonFilePath	: T_MaxString;
	sMlSvrNetId			: T_MaxString := 'local';
	eExecutionProvider	: E_ExecutionProvider := E_ExecutionProvider.CPU;
	bEnable				: BOOL;
	bReset					: BOOL;
	bLoadModel			: BOOL;
	nConfigureTimeout	: UDINT := 1000;
	nPredictTimeout		: UDINT := 100;
	nPriority			: UDINT := 0;
	fTheta					: REAL;
	fThetaDot				: REAL;
	fTorque				: REAL;
	fTemperature			: REAL;
	fDirectionFlag		: REAL;
	fThetaStep			: REAL := 0.25;
END_VAR
VAR
	fbMlSvr				: FB_MlSvrPrediction;
	stModelInput		: ST_ResidualHarmonicLstmSequenceDense360Input;
	stModelOutput		: ST_ResidualHarmonicLstmSequenceDense360Output;
	rtrig_model			: R_TRIG;
	nState					: INT := 0;
	nSequenceIndex		: INT;
	nOutputIndex		: INT;
END_VAR
VAR_OUTPUT
	bConfigured			: BOOL;
	bBusy					: BOOL;
	bPredictionPending	: BOOL;
	bPredictionReady	: BOOL;
	bResetDone			: BOOL;
	bError					: BOOL;
	nErrorCode			: HRESULT;
	nMaxInferenceDuration	: UDINT;
	aPredictionOutput	: ARRAY[0..8] OF REAL;
END_VAR

rtrig_model(CLK := bLoadModel);

IF rtrig_model.Q THEN
	bPredictionPending := FALSE;
	bPredictionReady := FALSE;
	bResetDone := FALSE;
	bError := FALSE;
	IF fbMlSvr.bConfigured THEN
		nState := 5;
	ELSE
		bConfigured := FALSE;
		nState := 10;
	END_IF
END_IF

IF bReset THEN
	bPredictionPending := FALSE;
	bPredictionReady := FALSE;
	bError := FALSE;
	IF fbMlSvr.bConfigured THEN
		nState := 5;
	ELSE
		bConfigured := FALSE;
		bResetDone := TRUE;
		nState := 0;
	END_IF
END_IF

CASE nState OF
	0:
		bBusy := FALSE;
		IF bLoadModel AND NOT(bConfigured) AND NOT(bReset) THEN
			nState := 10;
		END_IF

	5:
		bBusy := TRUE;
		IF fbMlSvr.Deconfigure(nTimeout := nConfigureTimeout) THEN
			nErrorCode := fbMlSvr.nErrorCode;
			bError := fbMlSvr.bError OR (nErrorCode <> 0);
			bConfigured := FALSE;
			bBusy := FALSE;
			bResetDone := NOT(bError);
			IF bError THEN
				nState := 90;
			ELSIF bReset THEN
				nState := 0;
			ELSE
				nState := 10;
			END_IF
		END_IF

	10:
		bBusy := TRUE;
		fbMlSvr.stPredictionParameter.sMlModelFilePath := sModelJsonFilePath;
		fbMlSvr.stPredictionParameter.sMlSvrNetId := sMlSvrNetId;
		fbMlSvr.stPredictionParameter.eExecutionProvider := eExecutionProvider;
		IF fbMlSvr.Configure(nTimeout := nConfigureTimeout, nPriority := nPriority) THEN
			nErrorCode := fbMlSvr.nErrorCode;
			bError := fbMlSvr.bError OR (nErrorCode <> 0);
			bConfigured := fbMlSvr.bConfigured AND NOT(bError);
			bBusy := FALSE;
			IF bConfigured THEN
				nState := 20;
			ELSE
				nState := 90;
			END_IF
		END_IF

	20:
		bBusy := FALSE;
		bPredictionPending := FALSE;
		IF bEnable AND bConfigured AND NOT(bError) AND NOT(bReset) THEN
			FOR nSequenceIndex := 0 TO 32 DO
				stModelInput.in_input_tensor[0,nSequenceIndex,0] := fTheta + (INT_TO_REAL(nSequenceIndex) * fThetaStep);
				stModelInput.in_input_tensor[0,nSequenceIndex,1] := fThetaDot;
				stModelInput.in_input_tensor[0,nSequenceIndex,2] := fTorque;
				stModelInput.in_input_tensor[0,nSequenceIndex,3] := fTemperature;
				stModelInput.in_input_tensor[0,nSequenceIndex,4] := fDirectionFlag;
			END_FOR
			bPredictionReady := FALSE;
			bPredictionPending := TRUE;
			nState := 30;
		END_IF

	30:
		bBusy := TRUE;
		bPredictionPending := TRUE;
		IF fbMlSvr.Predict(
			pDataIn := ADR(stModelInput),
			nDataInSize := SIZEOF(ST_ResidualHarmonicLstmSequenceDense360Input),
			pDataOut := ADR(stModelOutput),
			nDataOutSize := SIZEOF(ST_ResidualHarmonicLstmSequenceDense360Output),
			nTimeout := nPredictTimeout,
			nPriority := nPriority) THEN
			nErrorCode := fbMlSvr.nErrorCode;
			bError := fbMlSvr.bError OR (nErrorCode <> 0);
			nMaxInferenceDuration := fbMlSvr.nMaxInferenceDuration;
			bPredictionPending := FALSE;
			bBusy := FALSE;
			IF NOT(bError) THEN
				aPredictionOutput[0] := stModelOutput.out_prediction_tensor[0,0];
				FOR nOutputIndex := 1 TO 8 DO
					aPredictionOutput[nOutputIndex] := 0.0;
				END_FOR
				bPredictionReady := TRUE;
				nState := 20;
			ELSE
				nState := 90;
			END_IF
		END_IF

	90:
		bBusy := FALSE;
		bPredictionPending := FALSE;
		bError := TRUE;
END_CASE

nErrorCode := fbMlSvr.nErrorCode;
nMaxInferenceDuration := fbMlSvr.nMaxInferenceDuration;

END_FUNCTION_BLOCK

// ---- POUs/FB_ResidualHarmonicLstmSequenceSparseRcimTf3820Runner.TcPOU
FUNCTION_BLOCK FB_ResidualHarmonicLstmSequenceSparseRcimTf3820Runner
VAR_INPUT
	sModelJsonFilePath	: T_MaxString;
	sMlSvrNetId			: T_MaxString := 'local';
	eExecutionProvider	: E_ExecutionProvider := E_ExecutionProvider.CPU;
	bEnable				: BOOL;
	bReset					: BOOL;
	bLoadModel			: BOOL;
	nConfigureTimeout	: UDINT := 1000;
	nPredictTimeout		: UDINT := 100;
	nPriority			: UDINT := 0;
	fTheta					: REAL;
	fThetaDot				: REAL;
	fTorque				: REAL;
	fTemperature			: REAL;
	fDirectionFlag		: REAL;
	fThetaStep			: REAL := 0.25;
END_VAR
VAR
	fbMlSvr				: FB_MlSvrPrediction;
	stModelInput		: ST_ResidualHarmonicLstmSequenceSparseRcimInput;
	stModelOutput		: ST_ResidualHarmonicLstmSequenceSparseRcimOutput;
	rtrig_model			: R_TRIG;
	nState					: INT := 0;
	nSequenceIndex		: INT;
	nOutputIndex		: INT;
END_VAR
VAR_OUTPUT
	bConfigured			: BOOL;
	bBusy					: BOOL;
	bPredictionPending	: BOOL;
	bPredictionReady	: BOOL;
	bResetDone			: BOOL;
	bError					: BOOL;
	nErrorCode			: HRESULT;
	nMaxInferenceDuration	: UDINT;
	aPredictionOutput	: ARRAY[0..8] OF REAL;
END_VAR

rtrig_model(CLK := bLoadModel);

IF rtrig_model.Q THEN
	bPredictionPending := FALSE;
	bPredictionReady := FALSE;
	bResetDone := FALSE;
	bError := FALSE;
	IF fbMlSvr.bConfigured THEN
		nState := 5;
	ELSE
		bConfigured := FALSE;
		nState := 10;
	END_IF
END_IF

IF bReset THEN
	bPredictionPending := FALSE;
	bPredictionReady := FALSE;
	bError := FALSE;
	IF fbMlSvr.bConfigured THEN
		nState := 5;
	ELSE
		bConfigured := FALSE;
		bResetDone := TRUE;
		nState := 0;
	END_IF
END_IF

CASE nState OF
	0:
		bBusy := FALSE;
		IF bLoadModel AND NOT(bConfigured) AND NOT(bReset) THEN
			nState := 10;
		END_IF

	5:
		bBusy := TRUE;
		IF fbMlSvr.Deconfigure(nTimeout := nConfigureTimeout) THEN
			nErrorCode := fbMlSvr.nErrorCode;
			bError := fbMlSvr.bError OR (nErrorCode <> 0);
			bConfigured := FALSE;
			bBusy := FALSE;
			bResetDone := NOT(bError);
			IF bError THEN
				nState := 90;
			ELSIF bReset THEN
				nState := 0;
			ELSE
				nState := 10;
			END_IF
		END_IF

	10:
		bBusy := TRUE;
		fbMlSvr.stPredictionParameter.sMlModelFilePath := sModelJsonFilePath;
		fbMlSvr.stPredictionParameter.sMlSvrNetId := sMlSvrNetId;
		fbMlSvr.stPredictionParameter.eExecutionProvider := eExecutionProvider;
		IF fbMlSvr.Configure(nTimeout := nConfigureTimeout, nPriority := nPriority) THEN
			nErrorCode := fbMlSvr.nErrorCode;
			bError := fbMlSvr.bError OR (nErrorCode <> 0);
			bConfigured := fbMlSvr.bConfigured AND NOT(bError);
			bBusy := FALSE;
			IF bConfigured THEN
				nState := 20;
			ELSE
				nState := 90;
			END_IF
		END_IF

	20:
		bBusy := FALSE;
		bPredictionPending := FALSE;
		IF bEnable AND bConfigured AND NOT(bError) AND NOT(bReset) THEN
			FOR nSequenceIndex := 0 TO 32 DO
				stModelInput.in_input_tensor[0,nSequenceIndex,0] := fTheta + (INT_TO_REAL(nSequenceIndex) * fThetaStep);
				stModelInput.in_input_tensor[0,nSequenceIndex,1] := fThetaDot;
				stModelInput.in_input_tensor[0,nSequenceIndex,2] := fTorque;
				stModelInput.in_input_tensor[0,nSequenceIndex,3] := fTemperature;
				stModelInput.in_input_tensor[0,nSequenceIndex,4] := fDirectionFlag;
			END_FOR
			bPredictionReady := FALSE;
			bPredictionPending := TRUE;
			nState := 30;
		END_IF

	30:
		bBusy := TRUE;
		bPredictionPending := TRUE;
		IF fbMlSvr.Predict(
			pDataIn := ADR(stModelInput),
			nDataInSize := SIZEOF(ST_ResidualHarmonicLstmSequenceSparseRcimInput),
			pDataOut := ADR(stModelOutput),
			nDataOutSize := SIZEOF(ST_ResidualHarmonicLstmSequenceSparseRcimOutput),
			nTimeout := nPredictTimeout,
			nPriority := nPriority) THEN
			nErrorCode := fbMlSvr.nErrorCode;
			bError := fbMlSvr.bError OR (nErrorCode <> 0);
			nMaxInferenceDuration := fbMlSvr.nMaxInferenceDuration;
			bPredictionPending := FALSE;
			bBusy := FALSE;
			IF NOT(bError) THEN
				aPredictionOutput[0] := stModelOutput.out_prediction_tensor[0,0];
				FOR nOutputIndex := 1 TO 8 DO
					aPredictionOutput[nOutputIndex] := 0.0;
				END_FOR
				bPredictionReady := TRUE;
				nState := 20;
			ELSE
				nState := 90;
			END_IF
		END_IF

	90:
		bBusy := FALSE;
		bPredictionPending := FALSE;
		bError := TRUE;
END_CASE

nErrorCode := fbMlSvr.nErrorCode;
nMaxInferenceDuration := fbMlSvr.nMaxInferenceDuration;

END_FUNCTION_BLOCK

// ---- POUs/FB_ResidualHarmonicMlpTf3820Runner.TcPOU
FUNCTION_BLOCK FB_ResidualHarmonicMlpTf3820Runner
VAR_INPUT
	sModelJsonFilePath	: T_MaxString;
	sMlSvrNetId			: T_MaxString := 'local';
	eExecutionProvider	: E_ExecutionProvider := E_ExecutionProvider.CPU;
	bEnable				: BOOL;
	bReset					: BOOL;
	bLoadModel			: BOOL;
	nConfigureTimeout	: UDINT := 1000;
	nPredictTimeout		: UDINT := 100;
	nPriority			: UDINT := 0;
	fTheta					: REAL;
	fThetaDot				: REAL;
	fTorque				: REAL;
	fTemperature			: REAL;
	fDirectionFlag		: REAL;
	fThetaStep			: REAL := 0.25;
END_VAR
VAR
	fbMlSvr				: FB_MlSvrPrediction;
	stModelInput		: ST_ResidualHarmonicMlpInput;
	stModelOutput		: ST_ResidualHarmonicMlpOutput;
	rtrig_model			: R_TRIG;
	nState					: INT := 0;
	nSequenceIndex		: INT;
	nOutputIndex		: INT;
END_VAR
VAR_OUTPUT
	bConfigured			: BOOL;
	bBusy					: BOOL;
	bPredictionPending	: BOOL;
	bPredictionReady	: BOOL;
	bResetDone			: BOOL;
	bError					: BOOL;
	nErrorCode			: HRESULT;
	nMaxInferenceDuration	: UDINT;
	aPredictionOutput	: ARRAY[0..8] OF REAL;
END_VAR

rtrig_model(CLK := bLoadModel);

IF rtrig_model.Q THEN
	bPredictionPending := FALSE;
	bPredictionReady := FALSE;
	bResetDone := FALSE;
	bError := FALSE;
	IF fbMlSvr.bConfigured THEN
		nState := 5;
	ELSE
		bConfigured := FALSE;
		nState := 10;
	END_IF
END_IF

IF bReset THEN
	bPredictionPending := FALSE;
	bPredictionReady := FALSE;
	bError := FALSE;
	IF fbMlSvr.bConfigured THEN
		nState := 5;
	ELSE
		bConfigured := FALSE;
		bResetDone := TRUE;
		nState := 0;
	END_IF
END_IF

CASE nState OF
	0:
		bBusy := FALSE;
		IF bLoadModel AND NOT(bConfigured) AND NOT(bReset) THEN
			nState := 10;
		END_IF

	5:
		bBusy := TRUE;
		IF fbMlSvr.Deconfigure(nTimeout := nConfigureTimeout) THEN
			nErrorCode := fbMlSvr.nErrorCode;
			bError := fbMlSvr.bError OR (nErrorCode <> 0);
			bConfigured := FALSE;
			bBusy := FALSE;
			bResetDone := NOT(bError);
			IF bError THEN
				nState := 90;
			ELSIF bReset THEN
				nState := 0;
			ELSE
				nState := 10;
			END_IF
		END_IF

	10:
		bBusy := TRUE;
		fbMlSvr.stPredictionParameter.sMlModelFilePath := sModelJsonFilePath;
		fbMlSvr.stPredictionParameter.sMlSvrNetId := sMlSvrNetId;
		fbMlSvr.stPredictionParameter.eExecutionProvider := eExecutionProvider;
		IF fbMlSvr.Configure(nTimeout := nConfigureTimeout, nPriority := nPriority) THEN
			nErrorCode := fbMlSvr.nErrorCode;
			bError := fbMlSvr.bError OR (nErrorCode <> 0);
			bConfigured := fbMlSvr.bConfigured AND NOT(bError);
			bBusy := FALSE;
			IF bConfigured THEN
				nState := 20;
			ELSE
				nState := 90;
			END_IF
		END_IF

	20:
		bBusy := FALSE;
		bPredictionPending := FALSE;
		IF bEnable AND bConfigured AND NOT(bError) AND NOT(bReset) THEN
			stModelInput.in_input_tensor[0,0] := fTheta;
			stModelInput.in_input_tensor[0,1] := fThetaDot;
			stModelInput.in_input_tensor[0,2] := fTorque;
			stModelInput.in_input_tensor[0,3] := fTemperature;
			stModelInput.in_input_tensor[0,4] := fDirectionFlag;
			bPredictionReady := FALSE;
			bPredictionPending := TRUE;
			nState := 30;
		END_IF

	30:
		bBusy := TRUE;
		bPredictionPending := TRUE;
		IF fbMlSvr.Predict(
			pDataIn := ADR(stModelInput),
			nDataInSize := SIZEOF(ST_ResidualHarmonicMlpInput),
			pDataOut := ADR(stModelOutput),
			nDataOutSize := SIZEOF(ST_ResidualHarmonicMlpOutput),
			nTimeout := nPredictTimeout,
			nPriority := nPriority) THEN
			nErrorCode := fbMlSvr.nErrorCode;
			bError := fbMlSvr.bError OR (nErrorCode <> 0);
			nMaxInferenceDuration := fbMlSvr.nMaxInferenceDuration;
			bPredictionPending := FALSE;
			bBusy := FALSE;
			IF NOT(bError) THEN
				aPredictionOutput[0] := stModelOutput.out_prediction_tensor[0,0];
				FOR nOutputIndex := 1 TO 8 DO
					aPredictionOutput[nOutputIndex] := 0.0;
				END_FOR
				bPredictionReady := TRUE;
				nState := 20;
			ELSE
				nState := 90;
			END_IF
		END_IF

	90:
		bBusy := FALSE;
		bPredictionPending := FALSE;
		bError := TRUE;
END_CASE

nErrorCode := fbMlSvr.nErrorCode;
nMaxInferenceDuration := fbMlSvr.nMaxInferenceDuration;

END_FUNCTION_BLOCK

// ---- POUs/FB_TemporalConvolutionTf3820Runner.TcPOU
FUNCTION_BLOCK FB_TemporalConvolutionTf3820Runner
VAR_INPUT
	sModelJsonFilePath	: T_MaxString;
	sMlSvrNetId			: T_MaxString := 'local';
	eExecutionProvider	: E_ExecutionProvider := E_ExecutionProvider.CPU;
	bEnable				: BOOL;
	bReset					: BOOL;
	bLoadModel			: BOOL;
	nConfigureTimeout	: UDINT := 1000;
	nPredictTimeout		: UDINT := 100;
	nPriority			: UDINT := 0;
	fTheta					: REAL;
	fThetaDot				: REAL;
	fTorque				: REAL;
	fTemperature			: REAL;
	fDirectionFlag		: REAL;
	fThetaStep			: REAL := 0.25;
END_VAR
VAR
	fbMlSvr				: FB_MlSvrPrediction;
	stModelInput		: ST_TemporalConvolutionInput;
	stModelOutput		: ST_TemporalConvolutionOutput;
	rtrig_model			: R_TRIG;
	nState					: INT := 0;
	nSequenceIndex		: INT;
	nOutputIndex		: INT;
END_VAR
VAR_OUTPUT
	bConfigured			: BOOL;
	bBusy					: BOOL;
	bPredictionPending	: BOOL;
	bPredictionReady	: BOOL;
	bResetDone			: BOOL;
	bError					: BOOL;
	nErrorCode			: HRESULT;
	nMaxInferenceDuration	: UDINT;
	aPredictionOutput	: ARRAY[0..8] OF REAL;
END_VAR

rtrig_model(CLK := bLoadModel);

IF rtrig_model.Q THEN
	bPredictionPending := FALSE;
	bPredictionReady := FALSE;
	bResetDone := FALSE;
	bError := FALSE;
	IF fbMlSvr.bConfigured THEN
		nState := 5;
	ELSE
		bConfigured := FALSE;
		nState := 10;
	END_IF
END_IF

IF bReset THEN
	bPredictionPending := FALSE;
	bPredictionReady := FALSE;
	bError := FALSE;
	IF fbMlSvr.bConfigured THEN
		nState := 5;
	ELSE
		bConfigured := FALSE;
		bResetDone := TRUE;
		nState := 0;
	END_IF
END_IF

CASE nState OF
	0:
		bBusy := FALSE;
		IF bLoadModel AND NOT(bConfigured) AND NOT(bReset) THEN
			nState := 10;
		END_IF

	5:
		bBusy := TRUE;
		IF fbMlSvr.Deconfigure(nTimeout := nConfigureTimeout) THEN
			nErrorCode := fbMlSvr.nErrorCode;
			bError := fbMlSvr.bError OR (nErrorCode <> 0);
			bConfigured := FALSE;
			bBusy := FALSE;
			bResetDone := NOT(bError);
			IF bError THEN
				nState := 90;
			ELSIF bReset THEN
				nState := 0;
			ELSE
				nState := 10;
			END_IF
		END_IF

	10:
		bBusy := TRUE;
		fbMlSvr.stPredictionParameter.sMlModelFilePath := sModelJsonFilePath;
		fbMlSvr.stPredictionParameter.sMlSvrNetId := sMlSvrNetId;
		fbMlSvr.stPredictionParameter.eExecutionProvider := eExecutionProvider;
		IF fbMlSvr.Configure(nTimeout := nConfigureTimeout, nPriority := nPriority) THEN
			nErrorCode := fbMlSvr.nErrorCode;
			bError := fbMlSvr.bError OR (nErrorCode <> 0);
			bConfigured := fbMlSvr.bConfigured AND NOT(bError);
			bBusy := FALSE;
			IF bConfigured THEN
				nState := 20;
			ELSE
				nState := 90;
			END_IF
		END_IF

	20:
		bBusy := FALSE;
		bPredictionPending := FALSE;
		IF bEnable AND bConfigured AND NOT(bError) AND NOT(bReset) THEN
			FOR nSequenceIndex := 0 TO 32 DO
				stModelInput.in_input_tensor[0,nSequenceIndex,0] := fTheta + (INT_TO_REAL(nSequenceIndex) * fThetaStep);
				stModelInput.in_input_tensor[0,nSequenceIndex,1] := fThetaDot;
				stModelInput.in_input_tensor[0,nSequenceIndex,2] := fTorque;
				stModelInput.in_input_tensor[0,nSequenceIndex,3] := fTemperature;
				stModelInput.in_input_tensor[0,nSequenceIndex,4] := fDirectionFlag;
			END_FOR
			bPredictionReady := FALSE;
			bPredictionPending := TRUE;
			nState := 30;
		END_IF

	30:
		bBusy := TRUE;
		bPredictionPending := TRUE;
		IF fbMlSvr.Predict(
			pDataIn := ADR(stModelInput),
			nDataInSize := SIZEOF(ST_TemporalConvolutionInput),
			pDataOut := ADR(stModelOutput),
			nDataOutSize := SIZEOF(ST_TemporalConvolutionOutput),
			nTimeout := nPredictTimeout,
			nPriority := nPriority) THEN
			nErrorCode := fbMlSvr.nErrorCode;
			bError := fbMlSvr.bError OR (nErrorCode <> 0);
			nMaxInferenceDuration := fbMlSvr.nMaxInferenceDuration;
			bPredictionPending := FALSE;
			bBusy := FALSE;
			IF NOT(bError) THEN
				aPredictionOutput[0] := stModelOutput.out_prediction_tensor[0,0];
				FOR nOutputIndex := 1 TO 8 DO
					aPredictionOutput[nOutputIndex] := 0.0;
				END_FOR
				bPredictionReady := TRUE;
				nState := 20;
			ELSE
				nState := 90;
			END_IF
		END_IF

	90:
		bBusy := FALSE;
		bPredictionPending := FALSE;
		bError := TRUE;
END_CASE

nErrorCode := fbMlSvr.nErrorCode;
nMaxInferenceDuration := fbMlSvr.nMaxInferenceDuration;

END_FUNCTION_BLOCK

// ---- POUs/FB_TreeTf3820Runner.TcPOU
FUNCTION_BLOCK FB_TreeTf3820Runner
VAR_INPUT
	sModelJsonFilePath	: T_MaxString;
	sMlSvrNetId			: T_MaxString := 'local';
	eExecutionProvider	: E_ExecutionProvider := E_ExecutionProvider.CPU;
	bEnable				: BOOL;
	bReset					: BOOL;
	bLoadModel			: BOOL;
	nConfigureTimeout	: UDINT := 1000;
	nPredictTimeout		: UDINT := 100;
	nPriority			: UDINT := 0;
	fTheta					: REAL;
	fThetaDot				: REAL;
	fTorque				: REAL;
	fTemperature			: REAL;
	fDirectionFlag		: REAL;
	fThetaStep			: REAL := 0.25;
END_VAR
VAR
	fbMlSvr				: FB_MlSvrPrediction;
	stModelInput		: ST_TreeInput;
	stModelOutput		: ST_TreeOutput;
	rtrig_model			: R_TRIG;
	nState					: INT := 0;
	nSequenceIndex		: INT;
	nOutputIndex		: INT;
END_VAR
VAR_OUTPUT
	bConfigured			: BOOL;
	bBusy					: BOOL;
	bPredictionPending	: BOOL;
	bPredictionReady	: BOOL;
	bResetDone			: BOOL;
	bError					: BOOL;
	nErrorCode			: HRESULT;
	nMaxInferenceDuration	: UDINT;
	aPredictionOutput	: ARRAY[0..8] OF REAL;
END_VAR

rtrig_model(CLK := bLoadModel);

IF rtrig_model.Q THEN
	bPredictionPending := FALSE;
	bPredictionReady := FALSE;
	bResetDone := FALSE;
	bError := FALSE;
	IF fbMlSvr.bConfigured THEN
		nState := 5;
	ELSE
		bConfigured := FALSE;
		nState := 10;
	END_IF
END_IF

IF bReset THEN
	bPredictionPending := FALSE;
	bPredictionReady := FALSE;
	bError := FALSE;
	IF fbMlSvr.bConfigured THEN
		nState := 5;
	ELSE
		bConfigured := FALSE;
		bResetDone := TRUE;
		nState := 0;
	END_IF
END_IF

CASE nState OF
	0:
		bBusy := FALSE;
		IF bLoadModel AND NOT(bConfigured) AND NOT(bReset) THEN
			nState := 10;
		END_IF

	5:
		bBusy := TRUE;
		IF fbMlSvr.Deconfigure(nTimeout := nConfigureTimeout) THEN
			nErrorCode := fbMlSvr.nErrorCode;
			bError := fbMlSvr.bError OR (nErrorCode <> 0);
			bConfigured := FALSE;
			bBusy := FALSE;
			bResetDone := NOT(bError);
			IF bError THEN
				nState := 90;
			ELSIF bReset THEN
				nState := 0;
			ELSE
				nState := 10;
			END_IF
		END_IF

	10:
		bBusy := TRUE;
		fbMlSvr.stPredictionParameter.sMlModelFilePath := sModelJsonFilePath;
		fbMlSvr.stPredictionParameter.sMlSvrNetId := sMlSvrNetId;
		fbMlSvr.stPredictionParameter.eExecutionProvider := eExecutionProvider;
		IF fbMlSvr.Configure(nTimeout := nConfigureTimeout, nPriority := nPriority) THEN
			nErrorCode := fbMlSvr.nErrorCode;
			bError := fbMlSvr.bError OR (nErrorCode <> 0);
			bConfigured := fbMlSvr.bConfigured AND NOT(bError);
			bBusy := FALSE;
			IF bConfigured THEN
				nState := 20;
			ELSE
				nState := 90;
			END_IF
		END_IF

	20:
		bBusy := FALSE;
		bPredictionPending := FALSE;
		IF bEnable AND bConfigured AND NOT(bError) AND NOT(bReset) THEN
			stModelInput.in_float_input[0,0] := fTheta;
			stModelInput.in_float_input[0,1] := fThetaDot;
			stModelInput.in_float_input[0,2] := fTorque;
			stModelInput.in_float_input[0,3] := fTemperature;
			stModelInput.in_float_input[0,4] := fDirectionFlag;
			bPredictionReady := FALSE;
			bPredictionPending := TRUE;
			nState := 30;
		END_IF

	30:
		bBusy := TRUE;
		bPredictionPending := TRUE;
		IF fbMlSvr.Predict(
			pDataIn := ADR(stModelInput),
			nDataInSize := SIZEOF(ST_TreeInput),
			pDataOut := ADR(stModelOutput),
			nDataOutSize := SIZEOF(ST_TreeOutput),
			nTimeout := nPredictTimeout,
			nPriority := nPriority) THEN
			nErrorCode := fbMlSvr.nErrorCode;
			bError := fbMlSvr.bError OR (nErrorCode <> 0);
			nMaxInferenceDuration := fbMlSvr.nMaxInferenceDuration;
			bPredictionPending := FALSE;
			bBusy := FALSE;
			IF NOT(bError) THEN
				aPredictionOutput[0] := stModelOutput.out_variable[0,0];
				FOR nOutputIndex := 1 TO 8 DO
					aPredictionOutput[nOutputIndex] := 0.0;
				END_FOR
				bPredictionReady := TRUE;
				nState := 20;
			ELSE
				nState := 90;
			END_IF
		END_IF

	90:
		bBusy := FALSE;
		bPredictionPending := FALSE;
		bError := TRUE;
END_CASE

nErrorCode := fbMlSvr.nErrorCode;
nMaxInferenceDuration := fbMlSvr.nMaxInferenceDuration;

END_FUNCTION_BLOCK

// ---- POUs/FB_Wave31SequentialResidualOffsetProbeTf3820Runner.TcPOU
FUNCTION_BLOCK FB_Wave31SequentialResidualOffsetProbeTf3820Runner
VAR_INPUT
	sModelJsonFilePath	: T_MaxString;
	sMlSvrNetId			: T_MaxString := 'local';
	eExecutionProvider	: E_ExecutionProvider := E_ExecutionProvider.CPU;
	bEnable				: BOOL;
	bReset					: BOOL;
	bLoadModel			: BOOL;
	nConfigureTimeout	: UDINT := 1000;
	nPredictTimeout		: UDINT := 100;
	nPriority			: UDINT := 0;
	fTheta					: REAL;
	fThetaDot				: REAL;
	fTorque				: REAL;
	fTemperature			: REAL;
	fDirectionFlag		: REAL;
	fThetaStep			: REAL := 0.25;
END_VAR
VAR
	fbMlSvr				: FB_MlSvrPrediction;
	stModelInput		: ST_Wave31SequentialResidualOffsetProbeInput;
	stModelOutput		: ST_Wave31SequentialResidualOffsetProbeOutput;
	rtrig_model			: R_TRIG;
	nState					: INT := 0;
	nSequenceIndex		: INT;
	nOutputIndex		: INT;
END_VAR
VAR_OUTPUT
	bConfigured			: BOOL;
	bBusy					: BOOL;
	bPredictionPending	: BOOL;
	bPredictionReady	: BOOL;
	bResetDone			: BOOL;
	bError					: BOOL;
	nErrorCode			: HRESULT;
	nMaxInferenceDuration	: UDINT;
	aPredictionOutput	: ARRAY[0..8] OF REAL;
END_VAR

rtrig_model(CLK := bLoadModel);

IF rtrig_model.Q THEN
	bPredictionPending := FALSE;
	bPredictionReady := FALSE;
	bResetDone := FALSE;
	bError := FALSE;
	IF fbMlSvr.bConfigured THEN
		nState := 5;
	ELSE
		bConfigured := FALSE;
		nState := 10;
	END_IF
END_IF

IF bReset THEN
	bPredictionPending := FALSE;
	bPredictionReady := FALSE;
	bError := FALSE;
	IF fbMlSvr.bConfigured THEN
		nState := 5;
	ELSE
		bConfigured := FALSE;
		bResetDone := TRUE;
		nState := 0;
	END_IF
END_IF

CASE nState OF
	0:
		bBusy := FALSE;
		IF bLoadModel AND NOT(bConfigured) AND NOT(bReset) THEN
			nState := 10;
		END_IF

	5:
		bBusy := TRUE;
		IF fbMlSvr.Deconfigure(nTimeout := nConfigureTimeout) THEN
			nErrorCode := fbMlSvr.nErrorCode;
			bError := fbMlSvr.bError OR (nErrorCode <> 0);
			bConfigured := FALSE;
			bBusy := FALSE;
			bResetDone := NOT(bError);
			IF bError THEN
				nState := 90;
			ELSIF bReset THEN
				nState := 0;
			ELSE
				nState := 10;
			END_IF
		END_IF

	10:
		bBusy := TRUE;
		fbMlSvr.stPredictionParameter.sMlModelFilePath := sModelJsonFilePath;
		fbMlSvr.stPredictionParameter.sMlSvrNetId := sMlSvrNetId;
		fbMlSvr.stPredictionParameter.eExecutionProvider := eExecutionProvider;
		IF fbMlSvr.Configure(nTimeout := nConfigureTimeout, nPriority := nPriority) THEN
			nErrorCode := fbMlSvr.nErrorCode;
			bError := fbMlSvr.bError OR (nErrorCode <> 0);
			bConfigured := fbMlSvr.bConfigured AND NOT(bError);
			bBusy := FALSE;
			IF bConfigured THEN
				nState := 20;
			ELSE
				nState := 90;
			END_IF
		END_IF

	20:
		bBusy := FALSE;
		bPredictionPending := FALSE;
		IF bEnable AND bConfigured AND NOT(bError) AND NOT(bReset) THEN
			FOR nSequenceIndex := 0 TO 32 DO
				stModelInput.in_input_tensor[0,nSequenceIndex,0] := fTheta + (INT_TO_REAL(nSequenceIndex) * fThetaStep);
				stModelInput.in_input_tensor[0,nSequenceIndex,1] := fThetaDot;
				stModelInput.in_input_tensor[0,nSequenceIndex,2] := fTorque;
				stModelInput.in_input_tensor[0,nSequenceIndex,3] := fTemperature;
				stModelInput.in_input_tensor[0,nSequenceIndex,4] := fDirectionFlag;
			END_FOR
			bPredictionReady := FALSE;
			bPredictionPending := TRUE;
			nState := 30;
		END_IF

	30:
		bBusy := TRUE;
		bPredictionPending := TRUE;
		IF fbMlSvr.Predict(
			pDataIn := ADR(stModelInput),
			nDataInSize := SIZEOF(ST_Wave31SequentialResidualOffsetProbeInput),
			pDataOut := ADR(stModelOutput),
			nDataOutSize := SIZEOF(ST_Wave31SequentialResidualOffsetProbeOutput),
			nTimeout := nPredictTimeout,
			nPriority := nPriority) THEN
			nErrorCode := fbMlSvr.nErrorCode;
			bError := fbMlSvr.bError OR (nErrorCode <> 0);
			nMaxInferenceDuration := fbMlSvr.nMaxInferenceDuration;
			bPredictionPending := FALSE;
			bBusy := FALSE;
			IF NOT(bError) THEN
				aPredictionOutput[0] := stModelOutput.out_prediction_tensor[0,0];
				FOR nOutputIndex := 1 TO 8 DO
					aPredictionOutput[nOutputIndex] := 0.0;
				END_FOR
				bPredictionReady := TRUE;
				nState := 20;
			ELSE
				nState := 90;
			END_IF
		END_IF

	90:
		bBusy := FALSE;
		bPredictionPending := FALSE;
		bError := TRUE;
END_CASE

nErrorCode := fbMlSvr.nErrorCode;
nMaxInferenceDuration := fbMlSvr.nMaxInferenceDuration;

END_FUNCTION_BLOCK

// ---- POUs/FB_Wave32CleanSequentialResidualOffsetTf3820Runner.TcPOU
FUNCTION_BLOCK FB_Wave32CleanSequentialResidualOffsetTf3820Runner
VAR_INPUT
	sModelJsonFilePath	: T_MaxString;
	sMlSvrNetId			: T_MaxString := 'local';
	eExecutionProvider	: E_ExecutionProvider := E_ExecutionProvider.CPU;
	bEnable				: BOOL;
	bReset					: BOOL;
	bLoadModel			: BOOL;
	nConfigureTimeout	: UDINT := 1000;
	nPredictTimeout		: UDINT := 100;
	nPriority			: UDINT := 0;
	fTheta					: REAL;
	fThetaDot				: REAL;
	fTorque				: REAL;
	fTemperature			: REAL;
	fDirectionFlag		: REAL;
	fThetaStep			: REAL := 0.25;
END_VAR
VAR
	fbMlSvr				: FB_MlSvrPrediction;
	stModelInput		: ST_Wave32CleanSequentialResidualOffsetInput;
	stModelOutput		: ST_Wave32CleanSequentialResidualOffsetOutput;
	rtrig_model			: R_TRIG;
	nState					: INT := 0;
	nSequenceIndex		: INT;
	nOutputIndex		: INT;
END_VAR
VAR_OUTPUT
	bConfigured			: BOOL;
	bBusy					: BOOL;
	bPredictionPending	: BOOL;
	bPredictionReady	: BOOL;
	bResetDone			: BOOL;
	bError					: BOOL;
	nErrorCode			: HRESULT;
	nMaxInferenceDuration	: UDINT;
	aPredictionOutput	: ARRAY[0..8] OF REAL;
END_VAR

rtrig_model(CLK := bLoadModel);

IF rtrig_model.Q THEN
	bPredictionPending := FALSE;
	bPredictionReady := FALSE;
	bResetDone := FALSE;
	bError := FALSE;
	IF fbMlSvr.bConfigured THEN
		nState := 5;
	ELSE
		bConfigured := FALSE;
		nState := 10;
	END_IF
END_IF

IF bReset THEN
	bPredictionPending := FALSE;
	bPredictionReady := FALSE;
	bError := FALSE;
	IF fbMlSvr.bConfigured THEN
		nState := 5;
	ELSE
		bConfigured := FALSE;
		bResetDone := TRUE;
		nState := 0;
	END_IF
END_IF

CASE nState OF
	0:
		bBusy := FALSE;
		IF bLoadModel AND NOT(bConfigured) AND NOT(bReset) THEN
			nState := 10;
		END_IF

	5:
		bBusy := TRUE;
		IF fbMlSvr.Deconfigure(nTimeout := nConfigureTimeout) THEN
			nErrorCode := fbMlSvr.nErrorCode;
			bError := fbMlSvr.bError OR (nErrorCode <> 0);
			bConfigured := FALSE;
			bBusy := FALSE;
			bResetDone := NOT(bError);
			IF bError THEN
				nState := 90;
			ELSIF bReset THEN
				nState := 0;
			ELSE
				nState := 10;
			END_IF
		END_IF

	10:
		bBusy := TRUE;
		fbMlSvr.stPredictionParameter.sMlModelFilePath := sModelJsonFilePath;
		fbMlSvr.stPredictionParameter.sMlSvrNetId := sMlSvrNetId;
		fbMlSvr.stPredictionParameter.eExecutionProvider := eExecutionProvider;
		IF fbMlSvr.Configure(nTimeout := nConfigureTimeout, nPriority := nPriority) THEN
			nErrorCode := fbMlSvr.nErrorCode;
			bError := fbMlSvr.bError OR (nErrorCode <> 0);
			bConfigured := fbMlSvr.bConfigured AND NOT(bError);
			bBusy := FALSE;
			IF bConfigured THEN
				nState := 20;
			ELSE
				nState := 90;
			END_IF
		END_IF

	20:
		bBusy := FALSE;
		bPredictionPending := FALSE;
		IF bEnable AND bConfigured AND NOT(bError) AND NOT(bReset) THEN
			FOR nSequenceIndex := 0 TO 32 DO
				stModelInput.in_input_tensor[0,nSequenceIndex,0] := fTheta + (INT_TO_REAL(nSequenceIndex) * fThetaStep);
				stModelInput.in_input_tensor[0,nSequenceIndex,1] := fThetaDot;
				stModelInput.in_input_tensor[0,nSequenceIndex,2] := fTorque;
				stModelInput.in_input_tensor[0,nSequenceIndex,3] := fTemperature;
			END_FOR
			bPredictionReady := FALSE;
			bPredictionPending := TRUE;
			nState := 30;
		END_IF

	30:
		bBusy := TRUE;
		bPredictionPending := TRUE;
		IF fbMlSvr.Predict(
			pDataIn := ADR(stModelInput),
			nDataInSize := SIZEOF(ST_Wave32CleanSequentialResidualOffsetInput),
			pDataOut := ADR(stModelOutput),
			nDataOutSize := SIZEOF(ST_Wave32CleanSequentialResidualOffsetOutput),
			nTimeout := nPredictTimeout,
			nPriority := nPriority) THEN
			nErrorCode := fbMlSvr.nErrorCode;
			bError := fbMlSvr.bError OR (nErrorCode <> 0);
			nMaxInferenceDuration := fbMlSvr.nMaxInferenceDuration;
			bPredictionPending := FALSE;
			bBusy := FALSE;
			IF NOT(bError) THEN
				aPredictionOutput[0] := stModelOutput.out_prediction_tensor[0,0];
				FOR nOutputIndex := 1 TO 8 DO
					aPredictionOutput[nOutputIndex] := 0.0;
				END_FOR
				bPredictionReady := TRUE;
				nState := 20;
			ELSE
				nState := 90;
			END_IF
		END_IF

	90:
		bBusy := FALSE;
		bPredictionPending := FALSE;
		bError := TRUE;
END_CASE

nErrorCode := fbMlSvr.nErrorCode;
nMaxInferenceDuration := fbMlSvr.nMaxInferenceDuration;

END_FUNCTION_BLOCK

// ---- POUs/FB_Wave32HarmonicResidualOffsetTf3820Runner.TcPOU
FUNCTION_BLOCK FB_Wave32HarmonicResidualOffsetTf3820Runner
VAR_INPUT
	sModelJsonFilePath	: T_MaxString;
	sMlSvrNetId			: T_MaxString := 'local';
	eExecutionProvider	: E_ExecutionProvider := E_ExecutionProvider.CPU;
	bEnable				: BOOL;
	bReset					: BOOL;
	bLoadModel			: BOOL;
	nConfigureTimeout	: UDINT := 1000;
	nPredictTimeout		: UDINT := 100;
	nPriority			: UDINT := 0;
	fTheta					: REAL;
	fThetaDot				: REAL;
	fTorque				: REAL;
	fTemperature			: REAL;
	fDirectionFlag		: REAL;
	fThetaStep			: REAL := 0.25;
END_VAR
VAR
	fbMlSvr				: FB_MlSvrPrediction;
	stModelInput		: ST_Wave32HarmonicResidualOffsetInput;
	stModelOutput		: ST_Wave32HarmonicResidualOffsetOutput;
	rtrig_model			: R_TRIG;
	nState					: INT := 0;
	nSequenceIndex		: INT;
	nOutputIndex		: INT;
END_VAR
VAR_OUTPUT
	bConfigured			: BOOL;
	bBusy					: BOOL;
	bPredictionPending	: BOOL;
	bPredictionReady	: BOOL;
	bResetDone			: BOOL;
	bError					: BOOL;
	nErrorCode			: HRESULT;
	nMaxInferenceDuration	: UDINT;
	aPredictionOutput	: ARRAY[0..8] OF REAL;
END_VAR

rtrig_model(CLK := bLoadModel);

IF rtrig_model.Q THEN
	bPredictionPending := FALSE;
	bPredictionReady := FALSE;
	bResetDone := FALSE;
	bError := FALSE;
	IF fbMlSvr.bConfigured THEN
		nState := 5;
	ELSE
		bConfigured := FALSE;
		nState := 10;
	END_IF
END_IF

IF bReset THEN
	bPredictionPending := FALSE;
	bPredictionReady := FALSE;
	bError := FALSE;
	IF fbMlSvr.bConfigured THEN
		nState := 5;
	ELSE
		bConfigured := FALSE;
		bResetDone := TRUE;
		nState := 0;
	END_IF
END_IF

CASE nState OF
	0:
		bBusy := FALSE;
		IF bLoadModel AND NOT(bConfigured) AND NOT(bReset) THEN
			nState := 10;
		END_IF

	5:
		bBusy := TRUE;
		IF fbMlSvr.Deconfigure(nTimeout := nConfigureTimeout) THEN
			nErrorCode := fbMlSvr.nErrorCode;
			bError := fbMlSvr.bError OR (nErrorCode <> 0);
			bConfigured := FALSE;
			bBusy := FALSE;
			bResetDone := NOT(bError);
			IF bError THEN
				nState := 90;
			ELSIF bReset THEN
				nState := 0;
			ELSE
				nState := 10;
			END_IF
		END_IF

	10:
		bBusy := TRUE;
		fbMlSvr.stPredictionParameter.sMlModelFilePath := sModelJsonFilePath;
		fbMlSvr.stPredictionParameter.sMlSvrNetId := sMlSvrNetId;
		fbMlSvr.stPredictionParameter.eExecutionProvider := eExecutionProvider;
		IF fbMlSvr.Configure(nTimeout := nConfigureTimeout, nPriority := nPriority) THEN
			nErrorCode := fbMlSvr.nErrorCode;
			bError := fbMlSvr.bError OR (nErrorCode <> 0);
			bConfigured := fbMlSvr.bConfigured AND NOT(bError);
			bBusy := FALSE;
			IF bConfigured THEN
				nState := 20;
			ELSE
				nState := 90;
			END_IF
		END_IF

	20:
		bBusy := FALSE;
		bPredictionPending := FALSE;
		IF bEnable AND bConfigured AND NOT(bError) AND NOT(bReset) THEN
			FOR nSequenceIndex := 0 TO 32 DO
				stModelInput.in_input_tensor[0,nSequenceIndex,0] := fTheta + (INT_TO_REAL(nSequenceIndex) * fThetaStep);
				stModelInput.in_input_tensor[0,nSequenceIndex,1] := fThetaDot;
				stModelInput.in_input_tensor[0,nSequenceIndex,2] := fTorque;
				stModelInput.in_input_tensor[0,nSequenceIndex,3] := fTemperature;
			END_FOR
			bPredictionReady := FALSE;
			bPredictionPending := TRUE;
			nState := 30;
		END_IF

	30:
		bBusy := TRUE;
		bPredictionPending := TRUE;
		IF fbMlSvr.Predict(
			pDataIn := ADR(stModelInput),
			nDataInSize := SIZEOF(ST_Wave32HarmonicResidualOffsetInput),
			pDataOut := ADR(stModelOutput),
			nDataOutSize := SIZEOF(ST_Wave32HarmonicResidualOffsetOutput),
			nTimeout := nPredictTimeout,
			nPriority := nPriority) THEN
			nErrorCode := fbMlSvr.nErrorCode;
			bError := fbMlSvr.bError OR (nErrorCode <> 0);
			nMaxInferenceDuration := fbMlSvr.nMaxInferenceDuration;
			bPredictionPending := FALSE;
			bBusy := FALSE;
			IF NOT(bError) THEN
				aPredictionOutput[0] := stModelOutput.out_prediction_tensor[0,0];
				FOR nOutputIndex := 1 TO 8 DO
					aPredictionOutput[nOutputIndex] := 0.0;
				END_FOR
				bPredictionReady := TRUE;
				nState := 20;
			ELSE
				nState := 90;
			END_IF
		END_IF

	90:
		bBusy := FALSE;
		bPredictionPending := FALSE;
		bError := TRUE;
END_CASE

nErrorCode := fbMlSvr.nErrorCode;
nMaxInferenceDuration := fbMlSvr.nMaxInferenceDuration;

END_FUNCTION_BLOCK

// ---- POUs/FB_Wave33CurveAwarePointwiseControlTf3820Runner.TcPOU
FUNCTION_BLOCK FB_Wave33CurveAwarePointwiseControlTf3820Runner
VAR_INPUT
	sModelJsonFilePath	: T_MaxString;
	sMlSvrNetId			: T_MaxString := 'local';
	eExecutionProvider	: E_ExecutionProvider := E_ExecutionProvider.CPU;
	bEnable				: BOOL;
	bReset					: BOOL;
	bLoadModel			: BOOL;
	nConfigureTimeout	: UDINT := 1000;
	nPredictTimeout		: UDINT := 100;
	nPriority			: UDINT := 0;
	fTheta					: REAL;
	fThetaDot				: REAL;
	fTorque				: REAL;
	fTemperature			: REAL;
	fDirectionFlag		: REAL;
	fThetaStep			: REAL := 0.25;
END_VAR
VAR
	fbMlSvr				: FB_MlSvrPrediction;
	stModelInput		: ST_Wave33CurveAwarePointwiseControlInput;
	stModelOutput		: ST_Wave33CurveAwarePointwiseControlOutput;
	rtrig_model			: R_TRIG;
	nState					: INT := 0;
	nSequenceIndex		: INT;
	nOutputIndex		: INT;
END_VAR
VAR_OUTPUT
	bConfigured			: BOOL;
	bBusy					: BOOL;
	bPredictionPending	: BOOL;
	bPredictionReady	: BOOL;
	bResetDone			: BOOL;
	bError					: BOOL;
	nErrorCode			: HRESULT;
	nMaxInferenceDuration	: UDINT;
	aPredictionOutput	: ARRAY[0..8] OF REAL;
END_VAR

rtrig_model(CLK := bLoadModel);

IF rtrig_model.Q THEN
	bPredictionPending := FALSE;
	bPredictionReady := FALSE;
	bResetDone := FALSE;
	bError := FALSE;
	IF fbMlSvr.bConfigured THEN
		nState := 5;
	ELSE
		bConfigured := FALSE;
		nState := 10;
	END_IF
END_IF

IF bReset THEN
	bPredictionPending := FALSE;
	bPredictionReady := FALSE;
	bError := FALSE;
	IF fbMlSvr.bConfigured THEN
		nState := 5;
	ELSE
		bConfigured := FALSE;
		bResetDone := TRUE;
		nState := 0;
	END_IF
END_IF

CASE nState OF
	0:
		bBusy := FALSE;
		IF bLoadModel AND NOT(bConfigured) AND NOT(bReset) THEN
			nState := 10;
		END_IF

	5:
		bBusy := TRUE;
		IF fbMlSvr.Deconfigure(nTimeout := nConfigureTimeout) THEN
			nErrorCode := fbMlSvr.nErrorCode;
			bError := fbMlSvr.bError OR (nErrorCode <> 0);
			bConfigured := FALSE;
			bBusy := FALSE;
			bResetDone := NOT(bError);
			IF bError THEN
				nState := 90;
			ELSIF bReset THEN
				nState := 0;
			ELSE
				nState := 10;
			END_IF
		END_IF

	10:
		bBusy := TRUE;
		fbMlSvr.stPredictionParameter.sMlModelFilePath := sModelJsonFilePath;
		fbMlSvr.stPredictionParameter.sMlSvrNetId := sMlSvrNetId;
		fbMlSvr.stPredictionParameter.eExecutionProvider := eExecutionProvider;
		IF fbMlSvr.Configure(nTimeout := nConfigureTimeout, nPriority := nPriority) THEN
			nErrorCode := fbMlSvr.nErrorCode;
			bError := fbMlSvr.bError OR (nErrorCode <> 0);
			bConfigured := fbMlSvr.bConfigured AND NOT(bError);
			bBusy := FALSE;
			IF bConfigured THEN
				nState := 20;
			ELSE
				nState := 90;
			END_IF
		END_IF

	20:
		bBusy := FALSE;
		bPredictionPending := FALSE;
		IF bEnable AND bConfigured AND NOT(bError) AND NOT(bReset) THEN
			FOR nSequenceIndex := 0 TO 32 DO
				stModelInput.in_input_tensor[0,nSequenceIndex,0] := fTheta + (INT_TO_REAL(nSequenceIndex) * fThetaStep);
				stModelInput.in_input_tensor[0,nSequenceIndex,1] := fThetaDot;
				stModelInput.in_input_tensor[0,nSequenceIndex,2] := fTorque;
				stModelInput.in_input_tensor[0,nSequenceIndex,3] := fTemperature;
			END_FOR
			bPredictionReady := FALSE;
			bPredictionPending := TRUE;
			nState := 30;
		END_IF

	30:
		bBusy := TRUE;
		bPredictionPending := TRUE;
		IF fbMlSvr.Predict(
			pDataIn := ADR(stModelInput),
			nDataInSize := SIZEOF(ST_Wave33CurveAwarePointwiseControlInput),
			pDataOut := ADR(stModelOutput),
			nDataOutSize := SIZEOF(ST_Wave33CurveAwarePointwiseControlOutput),
			nTimeout := nPredictTimeout,
			nPriority := nPriority) THEN
			nErrorCode := fbMlSvr.nErrorCode;
			bError := fbMlSvr.bError OR (nErrorCode <> 0);
			nMaxInferenceDuration := fbMlSvr.nMaxInferenceDuration;
			bPredictionPending := FALSE;
			bBusy := FALSE;
			IF NOT(bError) THEN
				aPredictionOutput[0] := stModelOutput.out_prediction_tensor[0,0];
				FOR nOutputIndex := 1 TO 8 DO
					aPredictionOutput[nOutputIndex] := 0.0;
				END_FOR
				bPredictionReady := TRUE;
				nState := 20;
			ELSE
				nState := 90;
			END_IF
		END_IF

	90:
		bBusy := FALSE;
		bPredictionPending := FALSE;
		bError := TRUE;
END_CASE

nErrorCode := fbMlSvr.nErrorCode;
nMaxInferenceDuration := fbMlSvr.nMaxInferenceDuration;

END_FUNCTION_BLOCK

// ---- POUs/FB_Wave33FullCurveCompositeTf3820Runner.TcPOU
FUNCTION_BLOCK FB_Wave33FullCurveCompositeTf3820Runner
VAR_INPUT
	sModelJsonFilePath	: T_MaxString;
	sMlSvrNetId			: T_MaxString := 'local';
	eExecutionProvider	: E_ExecutionProvider := E_ExecutionProvider.CPU;
	bEnable				: BOOL;
	bReset					: BOOL;
	bLoadModel			: BOOL;
	nConfigureTimeout	: UDINT := 1000;
	nPredictTimeout		: UDINT := 100;
	nPriority			: UDINT := 0;
	fTheta					: REAL;
	fThetaDot				: REAL;
	fTorque				: REAL;
	fTemperature			: REAL;
	fDirectionFlag		: REAL;
	fThetaStep			: REAL := 0.25;
END_VAR
VAR
	fbMlSvr				: FB_MlSvrPrediction;
	stModelInput		: ST_Wave33FullCurveCompositeInput;
	stModelOutput		: ST_Wave33FullCurveCompositeOutput;
	rtrig_model			: R_TRIG;
	nState					: INT := 0;
	nSequenceIndex		: INT;
	nOutputIndex		: INT;
END_VAR
VAR_OUTPUT
	bConfigured			: BOOL;
	bBusy					: BOOL;
	bPredictionPending	: BOOL;
	bPredictionReady	: BOOL;
	bResetDone			: BOOL;
	bError					: BOOL;
	nErrorCode			: HRESULT;
	nMaxInferenceDuration	: UDINT;
	aPredictionOutput	: ARRAY[0..8] OF REAL;
END_VAR

rtrig_model(CLK := bLoadModel);

IF rtrig_model.Q THEN
	bPredictionPending := FALSE;
	bPredictionReady := FALSE;
	bResetDone := FALSE;
	bError := FALSE;
	IF fbMlSvr.bConfigured THEN
		nState := 5;
	ELSE
		bConfigured := FALSE;
		nState := 10;
	END_IF
END_IF

IF bReset THEN
	bPredictionPending := FALSE;
	bPredictionReady := FALSE;
	bError := FALSE;
	IF fbMlSvr.bConfigured THEN
		nState := 5;
	ELSE
		bConfigured := FALSE;
		bResetDone := TRUE;
		nState := 0;
	END_IF
END_IF

CASE nState OF
	0:
		bBusy := FALSE;
		IF bLoadModel AND NOT(bConfigured) AND NOT(bReset) THEN
			nState := 10;
		END_IF

	5:
		bBusy := TRUE;
		IF fbMlSvr.Deconfigure(nTimeout := nConfigureTimeout) THEN
			nErrorCode := fbMlSvr.nErrorCode;
			bError := fbMlSvr.bError OR (nErrorCode <> 0);
			bConfigured := FALSE;
			bBusy := FALSE;
			bResetDone := NOT(bError);
			IF bError THEN
				nState := 90;
			ELSIF bReset THEN
				nState := 0;
			ELSE
				nState := 10;
			END_IF
		END_IF

	10:
		bBusy := TRUE;
		fbMlSvr.stPredictionParameter.sMlModelFilePath := sModelJsonFilePath;
		fbMlSvr.stPredictionParameter.sMlSvrNetId := sMlSvrNetId;
		fbMlSvr.stPredictionParameter.eExecutionProvider := eExecutionProvider;
		IF fbMlSvr.Configure(nTimeout := nConfigureTimeout, nPriority := nPriority) THEN
			nErrorCode := fbMlSvr.nErrorCode;
			bError := fbMlSvr.bError OR (nErrorCode <> 0);
			bConfigured := fbMlSvr.bConfigured AND NOT(bError);
			bBusy := FALSE;
			IF bConfigured THEN
				nState := 20;
			ELSE
				nState := 90;
			END_IF
		END_IF

	20:
		bBusy := FALSE;
		bPredictionPending := FALSE;
		IF bEnable AND bConfigured AND NOT(bError) AND NOT(bReset) THEN
			FOR nSequenceIndex := 0 TO 32 DO
				stModelInput.in_input_tensor[0,nSequenceIndex,0] := fTheta + (INT_TO_REAL(nSequenceIndex) * fThetaStep);
				stModelInput.in_input_tensor[0,nSequenceIndex,1] := fThetaDot;
				stModelInput.in_input_tensor[0,nSequenceIndex,2] := fTorque;
				stModelInput.in_input_tensor[0,nSequenceIndex,3] := fTemperature;
			END_FOR
			bPredictionReady := FALSE;
			bPredictionPending := TRUE;
			nState := 30;
		END_IF

	30:
		bBusy := TRUE;
		bPredictionPending := TRUE;
		IF fbMlSvr.Predict(
			pDataIn := ADR(stModelInput),
			nDataInSize := SIZEOF(ST_Wave33FullCurveCompositeInput),
			pDataOut := ADR(stModelOutput),
			nDataOutSize := SIZEOF(ST_Wave33FullCurveCompositeOutput),
			nTimeout := nPredictTimeout,
			nPriority := nPriority) THEN
			nErrorCode := fbMlSvr.nErrorCode;
			bError := fbMlSvr.bError OR (nErrorCode <> 0);
			nMaxInferenceDuration := fbMlSvr.nMaxInferenceDuration;
			bPredictionPending := FALSE;
			bBusy := FALSE;
			IF NOT(bError) THEN
				aPredictionOutput[0] := stModelOutput.out_prediction_tensor[0,0];
				FOR nOutputIndex := 1 TO 8 DO
					aPredictionOutput[nOutputIndex] := 0.0;
				END_FOR
				bPredictionReady := TRUE;
				nState := 20;
			ELSE
				nState := 90;
			END_IF
		END_IF

	90:
		bBusy := FALSE;
		bPredictionPending := FALSE;
		bError := TRUE;
END_CASE

nErrorCode := fbMlSvr.nErrorCode;
nMaxInferenceDuration := fbMlSvr.nMaxInferenceDuration;

END_FUNCTION_BLOCK

// ---- POUs/FB_Wave33RawCenteredShapeCurveAwareTf3820Runner.TcPOU
FUNCTION_BLOCK FB_Wave33RawCenteredShapeCurveAwareTf3820Runner
VAR_INPUT
	sModelJsonFilePath	: T_MaxString;
	sMlSvrNetId			: T_MaxString := 'local';
	eExecutionProvider	: E_ExecutionProvider := E_ExecutionProvider.CPU;
	bEnable				: BOOL;
	bReset					: BOOL;
	bLoadModel			: BOOL;
	nConfigureTimeout	: UDINT := 1000;
	nPredictTimeout		: UDINT := 100;
	nPriority			: UDINT := 0;
	fTheta					: REAL;
	fThetaDot				: REAL;
	fTorque				: REAL;
	fTemperature			: REAL;
	fDirectionFlag		: REAL;
	fThetaStep			: REAL := 0.25;
END_VAR
VAR
	fbMlSvr				: FB_MlSvrPrediction;
	stModelInput		: ST_Wave33RawCenteredShapeCurveAwareInput;
	stModelOutput		: ST_Wave33RawCenteredShapeCurveAwareOutput;
	rtrig_model			: R_TRIG;
	nState					: INT := 0;
	nSequenceIndex		: INT;
	nOutputIndex		: INT;
END_VAR
VAR_OUTPUT
	bConfigured			: BOOL;
	bBusy					: BOOL;
	bPredictionPending	: BOOL;
	bPredictionReady	: BOOL;
	bResetDone			: BOOL;
	bError					: BOOL;
	nErrorCode			: HRESULT;
	nMaxInferenceDuration	: UDINT;
	aPredictionOutput	: ARRAY[0..8] OF REAL;
END_VAR

rtrig_model(CLK := bLoadModel);

IF rtrig_model.Q THEN
	bPredictionPending := FALSE;
	bPredictionReady := FALSE;
	bResetDone := FALSE;
	bError := FALSE;
	IF fbMlSvr.bConfigured THEN
		nState := 5;
	ELSE
		bConfigured := FALSE;
		nState := 10;
	END_IF
END_IF

IF bReset THEN
	bPredictionPending := FALSE;
	bPredictionReady := FALSE;
	bError := FALSE;
	IF fbMlSvr.bConfigured THEN
		nState := 5;
	ELSE
		bConfigured := FALSE;
		bResetDone := TRUE;
		nState := 0;
	END_IF
END_IF

CASE nState OF
	0:
		bBusy := FALSE;
		IF bLoadModel AND NOT(bConfigured) AND NOT(bReset) THEN
			nState := 10;
		END_IF

	5:
		bBusy := TRUE;
		IF fbMlSvr.Deconfigure(nTimeout := nConfigureTimeout) THEN
			nErrorCode := fbMlSvr.nErrorCode;
			bError := fbMlSvr.bError OR (nErrorCode <> 0);
			bConfigured := FALSE;
			bBusy := FALSE;
			bResetDone := NOT(bError);
			IF bError THEN
				nState := 90;
			ELSIF bReset THEN
				nState := 0;
			ELSE
				nState := 10;
			END_IF
		END_IF

	10:
		bBusy := TRUE;
		fbMlSvr.stPredictionParameter.sMlModelFilePath := sModelJsonFilePath;
		fbMlSvr.stPredictionParameter.sMlSvrNetId := sMlSvrNetId;
		fbMlSvr.stPredictionParameter.eExecutionProvider := eExecutionProvider;
		IF fbMlSvr.Configure(nTimeout := nConfigureTimeout, nPriority := nPriority) THEN
			nErrorCode := fbMlSvr.nErrorCode;
			bError := fbMlSvr.bError OR (nErrorCode <> 0);
			bConfigured := fbMlSvr.bConfigured AND NOT(bError);
			bBusy := FALSE;
			IF bConfigured THEN
				nState := 20;
			ELSE
				nState := 90;
			END_IF
		END_IF

	20:
		bBusy := FALSE;
		bPredictionPending := FALSE;
		IF bEnable AND bConfigured AND NOT(bError) AND NOT(bReset) THEN
			FOR nSequenceIndex := 0 TO 32 DO
				stModelInput.in_input_tensor[0,nSequenceIndex,0] := fTheta + (INT_TO_REAL(nSequenceIndex) * fThetaStep);
				stModelInput.in_input_tensor[0,nSequenceIndex,1] := fThetaDot;
				stModelInput.in_input_tensor[0,nSequenceIndex,2] := fTorque;
				stModelInput.in_input_tensor[0,nSequenceIndex,3] := fTemperature;
			END_FOR
			bPredictionReady := FALSE;
			bPredictionPending := TRUE;
			nState := 30;
		END_IF

	30:
		bBusy := TRUE;
		bPredictionPending := TRUE;
		IF fbMlSvr.Predict(
			pDataIn := ADR(stModelInput),
			nDataInSize := SIZEOF(ST_Wave33RawCenteredShapeCurveAwareInput),
			pDataOut := ADR(stModelOutput),
			nDataOutSize := SIZEOF(ST_Wave33RawCenteredShapeCurveAwareOutput),
			nTimeout := nPredictTimeout,
			nPriority := nPriority) THEN
			nErrorCode := fbMlSvr.nErrorCode;
			bError := fbMlSvr.bError OR (nErrorCode <> 0);
			nMaxInferenceDuration := fbMlSvr.nMaxInferenceDuration;
			bPredictionPending := FALSE;
			bBusy := FALSE;
			IF NOT(bError) THEN
				aPredictionOutput[0] := stModelOutput.out_prediction_tensor[0,0];
				FOR nOutputIndex := 1 TO 8 DO
					aPredictionOutput[nOutputIndex] := 0.0;
				END_FOR
				bPredictionReady := TRUE;
				nState := 20;
			ELSE
				nState := 90;
			END_IF
		END_IF

	90:
		bBusy := FALSE;
		bPredictionPending := FALSE;
		bError := TRUE;
END_CASE

nErrorCode := fbMlSvr.nErrorCode;
nMaxInferenceDuration := fbMlSvr.nMaxInferenceDuration;

END_FUNCTION_BLOCK

// ---- POUs/FB_Wave33RawOffsetCurveAwareTf3820Runner.TcPOU
FUNCTION_BLOCK FB_Wave33RawOffsetCurveAwareTf3820Runner
VAR_INPUT
	sModelJsonFilePath	: T_MaxString;
	sMlSvrNetId			: T_MaxString := 'local';
	eExecutionProvider	: E_ExecutionProvider := E_ExecutionProvider.CPU;
	bEnable				: BOOL;
	bReset					: BOOL;
	bLoadModel			: BOOL;
	nConfigureTimeout	: UDINT := 1000;
	nPredictTimeout		: UDINT := 100;
	nPriority			: UDINT := 0;
	fTheta					: REAL;
	fThetaDot				: REAL;
	fTorque				: REAL;
	fTemperature			: REAL;
	fDirectionFlag		: REAL;
	fThetaStep			: REAL := 0.25;
END_VAR
VAR
	fbMlSvr				: FB_MlSvrPrediction;
	stModelInput		: ST_Wave33RawOffsetCurveAwareInput;
	stModelOutput		: ST_Wave33RawOffsetCurveAwareOutput;
	rtrig_model			: R_TRIG;
	nState					: INT := 0;
	nSequenceIndex		: INT;
	nOutputIndex		: INT;
END_VAR
VAR_OUTPUT
	bConfigured			: BOOL;
	bBusy					: BOOL;
	bPredictionPending	: BOOL;
	bPredictionReady	: BOOL;
	bResetDone			: BOOL;
	bError					: BOOL;
	nErrorCode			: HRESULT;
	nMaxInferenceDuration	: UDINT;
	aPredictionOutput	: ARRAY[0..8] OF REAL;
END_VAR

rtrig_model(CLK := bLoadModel);

IF rtrig_model.Q THEN
	bPredictionPending := FALSE;
	bPredictionReady := FALSE;
	bResetDone := FALSE;
	bError := FALSE;
	IF fbMlSvr.bConfigured THEN
		nState := 5;
	ELSE
		bConfigured := FALSE;
		nState := 10;
	END_IF
END_IF

IF bReset THEN
	bPredictionPending := FALSE;
	bPredictionReady := FALSE;
	bError := FALSE;
	IF fbMlSvr.bConfigured THEN
		nState := 5;
	ELSE
		bConfigured := FALSE;
		bResetDone := TRUE;
		nState := 0;
	END_IF
END_IF

CASE nState OF
	0:
		bBusy := FALSE;
		IF bLoadModel AND NOT(bConfigured) AND NOT(bReset) THEN
			nState := 10;
		END_IF

	5:
		bBusy := TRUE;
		IF fbMlSvr.Deconfigure(nTimeout := nConfigureTimeout) THEN
			nErrorCode := fbMlSvr.nErrorCode;
			bError := fbMlSvr.bError OR (nErrorCode <> 0);
			bConfigured := FALSE;
			bBusy := FALSE;
			bResetDone := NOT(bError);
			IF bError THEN
				nState := 90;
			ELSIF bReset THEN
				nState := 0;
			ELSE
				nState := 10;
			END_IF
		END_IF

	10:
		bBusy := TRUE;
		fbMlSvr.stPredictionParameter.sMlModelFilePath := sModelJsonFilePath;
		fbMlSvr.stPredictionParameter.sMlSvrNetId := sMlSvrNetId;
		fbMlSvr.stPredictionParameter.eExecutionProvider := eExecutionProvider;
		IF fbMlSvr.Configure(nTimeout := nConfigureTimeout, nPriority := nPriority) THEN
			nErrorCode := fbMlSvr.nErrorCode;
			bError := fbMlSvr.bError OR (nErrorCode <> 0);
			bConfigured := fbMlSvr.bConfigured AND NOT(bError);
			bBusy := FALSE;
			IF bConfigured THEN
				nState := 20;
			ELSE
				nState := 90;
			END_IF
		END_IF

	20:
		bBusy := FALSE;
		bPredictionPending := FALSE;
		IF bEnable AND bConfigured AND NOT(bError) AND NOT(bReset) THEN
			FOR nSequenceIndex := 0 TO 32 DO
				stModelInput.in_input_tensor[0,nSequenceIndex,0] := fTheta + (INT_TO_REAL(nSequenceIndex) * fThetaStep);
				stModelInput.in_input_tensor[0,nSequenceIndex,1] := fThetaDot;
				stModelInput.in_input_tensor[0,nSequenceIndex,2] := fTorque;
				stModelInput.in_input_tensor[0,nSequenceIndex,3] := fTemperature;
			END_FOR
			bPredictionReady := FALSE;
			bPredictionPending := TRUE;
			nState := 30;
		END_IF

	30:
		bBusy := TRUE;
		bPredictionPending := TRUE;
		IF fbMlSvr.Predict(
			pDataIn := ADR(stModelInput),
			nDataInSize := SIZEOF(ST_Wave33RawOffsetCurveAwareInput),
			pDataOut := ADR(stModelOutput),
			nDataOutSize := SIZEOF(ST_Wave33RawOffsetCurveAwareOutput),
			nTimeout := nPredictTimeout,
			nPriority := nPriority) THEN
			nErrorCode := fbMlSvr.nErrorCode;
			bError := fbMlSvr.bError OR (nErrorCode <> 0);
			nMaxInferenceDuration := fbMlSvr.nMaxInferenceDuration;
			bPredictionPending := FALSE;
			bBusy := FALSE;
			IF NOT(bError) THEN
				aPredictionOutput[0] := stModelOutput.out_prediction_tensor[0,0];
				FOR nOutputIndex := 1 TO 8 DO
					aPredictionOutput[nOutputIndex] := 0.0;
				END_FOR
				bPredictionReady := TRUE;
				nState := 20;
			ELSE
				nState := 90;
			END_IF
		END_IF

	90:
		bBusy := FALSE;
		bPredictionPending := FALSE;
		bError := TRUE;
END_CASE

nErrorCode := fbMlSvr.nErrorCode;
nMaxInferenceDuration := fbMlSvr.nMaxInferenceDuration;

END_FUNCTION_BLOCK

// ---- POUs/FB_Wave41LogCoshRobustLossTf3820Runner.TcPOU
FUNCTION_BLOCK FB_Wave41LogCoshRobustLossTf3820Runner
VAR_INPUT
	sModelJsonFilePath	: T_MaxString;
	sMlSvrNetId			: T_MaxString := 'local';
	eExecutionProvider	: E_ExecutionProvider := E_ExecutionProvider.CPU;
	bEnable				: BOOL;
	bReset					: BOOL;
	bLoadModel			: BOOL;
	nConfigureTimeout	: UDINT := 1000;
	nPredictTimeout		: UDINT := 100;
	nPriority			: UDINT := 0;
	fTheta					: REAL;
	fThetaDot				: REAL;
	fTorque				: REAL;
	fTemperature			: REAL;
	fDirectionFlag		: REAL;
	fThetaStep			: REAL := 0.25;
END_VAR
VAR
	fbMlSvr				: FB_MlSvrPrediction;
	stModelInput		: ST_Wave41LogCoshRobustLossInput;
	stModelOutput		: ST_Wave41LogCoshRobustLossOutput;
	rtrig_model			: R_TRIG;
	nState					: INT := 0;
	nSequenceIndex		: INT;
	nOutputIndex		: INT;
END_VAR
VAR_OUTPUT
	bConfigured			: BOOL;
	bBusy					: BOOL;
	bPredictionPending	: BOOL;
	bPredictionReady	: BOOL;
	bResetDone			: BOOL;
	bError					: BOOL;
	nErrorCode			: HRESULT;
	nMaxInferenceDuration	: UDINT;
	aPredictionOutput	: ARRAY[0..8] OF REAL;
END_VAR

rtrig_model(CLK := bLoadModel);

IF rtrig_model.Q THEN
	bPredictionPending := FALSE;
	bPredictionReady := FALSE;
	bResetDone := FALSE;
	bError := FALSE;
	IF fbMlSvr.bConfigured THEN
		nState := 5;
	ELSE
		bConfigured := FALSE;
		nState := 10;
	END_IF
END_IF

IF bReset THEN
	bPredictionPending := FALSE;
	bPredictionReady := FALSE;
	bError := FALSE;
	IF fbMlSvr.bConfigured THEN
		nState := 5;
	ELSE
		bConfigured := FALSE;
		bResetDone := TRUE;
		nState := 0;
	END_IF
END_IF

CASE nState OF
	0:
		bBusy := FALSE;
		IF bLoadModel AND NOT(bConfigured) AND NOT(bReset) THEN
			nState := 10;
		END_IF

	5:
		bBusy := TRUE;
		IF fbMlSvr.Deconfigure(nTimeout := nConfigureTimeout) THEN
			nErrorCode := fbMlSvr.nErrorCode;
			bError := fbMlSvr.bError OR (nErrorCode <> 0);
			bConfigured := FALSE;
			bBusy := FALSE;
			bResetDone := NOT(bError);
			IF bError THEN
				nState := 90;
			ELSIF bReset THEN
				nState := 0;
			ELSE
				nState := 10;
			END_IF
		END_IF

	10:
		bBusy := TRUE;
		fbMlSvr.stPredictionParameter.sMlModelFilePath := sModelJsonFilePath;
		fbMlSvr.stPredictionParameter.sMlSvrNetId := sMlSvrNetId;
		fbMlSvr.stPredictionParameter.eExecutionProvider := eExecutionProvider;
		IF fbMlSvr.Configure(nTimeout := nConfigureTimeout, nPriority := nPriority) THEN
			nErrorCode := fbMlSvr.nErrorCode;
			bError := fbMlSvr.bError OR (nErrorCode <> 0);
			bConfigured := fbMlSvr.bConfigured AND NOT(bError);
			bBusy := FALSE;
			IF bConfigured THEN
				nState := 20;
			ELSE
				nState := 90;
			END_IF
		END_IF

	20:
		bBusy := FALSE;
		bPredictionPending := FALSE;
		IF bEnable AND bConfigured AND NOT(bError) AND NOT(bReset) THEN
			FOR nSequenceIndex := 0 TO 32 DO
				stModelInput.in_input_tensor[0,nSequenceIndex,0] := fTheta + (INT_TO_REAL(nSequenceIndex) * fThetaStep);
				stModelInput.in_input_tensor[0,nSequenceIndex,1] := fThetaDot;
				stModelInput.in_input_tensor[0,nSequenceIndex,2] := fTorque;
				stModelInput.in_input_tensor[0,nSequenceIndex,3] := fTemperature;
			END_FOR
			bPredictionReady := FALSE;
			bPredictionPending := TRUE;
			nState := 30;
		END_IF

	30:
		bBusy := TRUE;
		bPredictionPending := TRUE;
		IF fbMlSvr.Predict(
			pDataIn := ADR(stModelInput),
			nDataInSize := SIZEOF(ST_Wave41LogCoshRobustLossInput),
			pDataOut := ADR(stModelOutput),
			nDataOutSize := SIZEOF(ST_Wave41LogCoshRobustLossOutput),
			nTimeout := nPredictTimeout,
			nPriority := nPriority) THEN
			nErrorCode := fbMlSvr.nErrorCode;
			bError := fbMlSvr.bError OR (nErrorCode <> 0);
			nMaxInferenceDuration := fbMlSvr.nMaxInferenceDuration;
			bPredictionPending := FALSE;
			bBusy := FALSE;
			IF NOT(bError) THEN
				aPredictionOutput[0] := stModelOutput.out_prediction_tensor[0,0];
				FOR nOutputIndex := 1 TO 8 DO
					aPredictionOutput[nOutputIndex] := 0.0;
				END_FOR
				bPredictionReady := TRUE;
				nState := 20;
			ELSE
				nState := 90;
			END_IF
		END_IF

	90:
		bBusy := FALSE;
		bPredictionPending := FALSE;
		bError := TRUE;
END_CASE

nErrorCode := fbMlSvr.nErrorCode;
nMaxInferenceDuration := fbMlSvr.nMaxInferenceDuration;

END_FUNCTION_BLOCK

// ---- POUs/FB_Wave41MaeRobustLossTf3820Runner.TcPOU
FUNCTION_BLOCK FB_Wave41MaeRobustLossTf3820Runner
VAR_INPUT
	sModelJsonFilePath	: T_MaxString;
	sMlSvrNetId			: T_MaxString := 'local';
	eExecutionProvider	: E_ExecutionProvider := E_ExecutionProvider.CPU;
	bEnable				: BOOL;
	bReset					: BOOL;
	bLoadModel			: BOOL;
	nConfigureTimeout	: UDINT := 1000;
	nPredictTimeout		: UDINT := 100;
	nPriority			: UDINT := 0;
	fTheta					: REAL;
	fThetaDot				: REAL;
	fTorque				: REAL;
	fTemperature			: REAL;
	fDirectionFlag		: REAL;
	fThetaStep			: REAL := 0.25;
END_VAR
VAR
	fbMlSvr				: FB_MlSvrPrediction;
	stModelInput		: ST_Wave41MaeRobustLossInput;
	stModelOutput		: ST_Wave41MaeRobustLossOutput;
	rtrig_model			: R_TRIG;
	nState					: INT := 0;
	nSequenceIndex		: INT;
	nOutputIndex		: INT;
END_VAR
VAR_OUTPUT
	bConfigured			: BOOL;
	bBusy					: BOOL;
	bPredictionPending	: BOOL;
	bPredictionReady	: BOOL;
	bResetDone			: BOOL;
	bError					: BOOL;
	nErrorCode			: HRESULT;
	nMaxInferenceDuration	: UDINT;
	aPredictionOutput	: ARRAY[0..8] OF REAL;
END_VAR

rtrig_model(CLK := bLoadModel);

IF rtrig_model.Q THEN
	bPredictionPending := FALSE;
	bPredictionReady := FALSE;
	bResetDone := FALSE;
	bError := FALSE;
	IF fbMlSvr.bConfigured THEN
		nState := 5;
	ELSE
		bConfigured := FALSE;
		nState := 10;
	END_IF
END_IF

IF bReset THEN
	bPredictionPending := FALSE;
	bPredictionReady := FALSE;
	bError := FALSE;
	IF fbMlSvr.bConfigured THEN
		nState := 5;
	ELSE
		bConfigured := FALSE;
		bResetDone := TRUE;
		nState := 0;
	END_IF
END_IF

CASE nState OF
	0:
		bBusy := FALSE;
		IF bLoadModel AND NOT(bConfigured) AND NOT(bReset) THEN
			nState := 10;
		END_IF

	5:
		bBusy := TRUE;
		IF fbMlSvr.Deconfigure(nTimeout := nConfigureTimeout) THEN
			nErrorCode := fbMlSvr.nErrorCode;
			bError := fbMlSvr.bError OR (nErrorCode <> 0);
			bConfigured := FALSE;
			bBusy := FALSE;
			bResetDone := NOT(bError);
			IF bError THEN
				nState := 90;
			ELSIF bReset THEN
				nState := 0;
			ELSE
				nState := 10;
			END_IF
		END_IF

	10:
		bBusy := TRUE;
		fbMlSvr.stPredictionParameter.sMlModelFilePath := sModelJsonFilePath;
		fbMlSvr.stPredictionParameter.sMlSvrNetId := sMlSvrNetId;
		fbMlSvr.stPredictionParameter.eExecutionProvider := eExecutionProvider;
		IF fbMlSvr.Configure(nTimeout := nConfigureTimeout, nPriority := nPriority) THEN
			nErrorCode := fbMlSvr.nErrorCode;
			bError := fbMlSvr.bError OR (nErrorCode <> 0);
			bConfigured := fbMlSvr.bConfigured AND NOT(bError);
			bBusy := FALSE;
			IF bConfigured THEN
				nState := 20;
			ELSE
				nState := 90;
			END_IF
		END_IF

	20:
		bBusy := FALSE;
		bPredictionPending := FALSE;
		IF bEnable AND bConfigured AND NOT(bError) AND NOT(bReset) THEN
			FOR nSequenceIndex := 0 TO 32 DO
				stModelInput.in_input_tensor[0,nSequenceIndex,0] := fTheta + (INT_TO_REAL(nSequenceIndex) * fThetaStep);
				stModelInput.in_input_tensor[0,nSequenceIndex,1] := fThetaDot;
				stModelInput.in_input_tensor[0,nSequenceIndex,2] := fTorque;
				stModelInput.in_input_tensor[0,nSequenceIndex,3] := fTemperature;
			END_FOR
			bPredictionReady := FALSE;
			bPredictionPending := TRUE;
			nState := 30;
		END_IF

	30:
		bBusy := TRUE;
		bPredictionPending := TRUE;
		IF fbMlSvr.Predict(
			pDataIn := ADR(stModelInput),
			nDataInSize := SIZEOF(ST_Wave41MaeRobustLossInput),
			pDataOut := ADR(stModelOutput),
			nDataOutSize := SIZEOF(ST_Wave41MaeRobustLossOutput),
			nTimeout := nPredictTimeout,
			nPriority := nPriority) THEN
			nErrorCode := fbMlSvr.nErrorCode;
			bError := fbMlSvr.bError OR (nErrorCode <> 0);
			nMaxInferenceDuration := fbMlSvr.nMaxInferenceDuration;
			bPredictionPending := FALSE;
			bBusy := FALSE;
			IF NOT(bError) THEN
				aPredictionOutput[0] := stModelOutput.out_prediction_tensor[0,0];
				FOR nOutputIndex := 1 TO 8 DO
					aPredictionOutput[nOutputIndex] := 0.0;
				END_FOR
				bPredictionReady := TRUE;
				nState := 20;
			ELSE
				nState := 90;
			END_IF
		END_IF

	90:
		bBusy := FALSE;
		bPredictionPending := FALSE;
		bError := TRUE;
END_CASE

nErrorCode := fbMlSvr.nErrorCode;
nMaxInferenceDuration := fbMlSvr.nMaxInferenceDuration;

END_FUNCTION_BLOCK

// ---- POUs/FB_Wave41SmoothL1RobustLossTf3820Runner.TcPOU
FUNCTION_BLOCK FB_Wave41SmoothL1RobustLossTf3820Runner
VAR_INPUT
	sModelJsonFilePath	: T_MaxString;
	sMlSvrNetId			: T_MaxString := 'local';
	eExecutionProvider	: E_ExecutionProvider := E_ExecutionProvider.CPU;
	bEnable				: BOOL;
	bReset					: BOOL;
	bLoadModel			: BOOL;
	nConfigureTimeout	: UDINT := 1000;
	nPredictTimeout		: UDINT := 100;
	nPriority			: UDINT := 0;
	fTheta					: REAL;
	fThetaDot				: REAL;
	fTorque				: REAL;
	fTemperature			: REAL;
	fDirectionFlag		: REAL;
	fThetaStep			: REAL := 0.25;
END_VAR
VAR
	fbMlSvr				: FB_MlSvrPrediction;
	stModelInput		: ST_Wave41SmoothL1RobustLossInput;
	stModelOutput		: ST_Wave41SmoothL1RobustLossOutput;
	rtrig_model			: R_TRIG;
	nState					: INT := 0;
	nSequenceIndex		: INT;
	nOutputIndex		: INT;
END_VAR
VAR_OUTPUT
	bConfigured			: BOOL;
	bBusy					: BOOL;
	bPredictionPending	: BOOL;
	bPredictionReady	: BOOL;
	bResetDone			: BOOL;
	bError					: BOOL;
	nErrorCode			: HRESULT;
	nMaxInferenceDuration	: UDINT;
	aPredictionOutput	: ARRAY[0..8] OF REAL;
END_VAR

rtrig_model(CLK := bLoadModel);

IF rtrig_model.Q THEN
	bPredictionPending := FALSE;
	bPredictionReady := FALSE;
	bResetDone := FALSE;
	bError := FALSE;
	IF fbMlSvr.bConfigured THEN
		nState := 5;
	ELSE
		bConfigured := FALSE;
		nState := 10;
	END_IF
END_IF

IF bReset THEN
	bPredictionPending := FALSE;
	bPredictionReady := FALSE;
	bError := FALSE;
	IF fbMlSvr.bConfigured THEN
		nState := 5;
	ELSE
		bConfigured := FALSE;
		bResetDone := TRUE;
		nState := 0;
	END_IF
END_IF

CASE nState OF
	0:
		bBusy := FALSE;
		IF bLoadModel AND NOT(bConfigured) AND NOT(bReset) THEN
			nState := 10;
		END_IF

	5:
		bBusy := TRUE;
		IF fbMlSvr.Deconfigure(nTimeout := nConfigureTimeout) THEN
			nErrorCode := fbMlSvr.nErrorCode;
			bError := fbMlSvr.bError OR (nErrorCode <> 0);
			bConfigured := FALSE;
			bBusy := FALSE;
			bResetDone := NOT(bError);
			IF bError THEN
				nState := 90;
			ELSIF bReset THEN
				nState := 0;
			ELSE
				nState := 10;
			END_IF
		END_IF

	10:
		bBusy := TRUE;
		fbMlSvr.stPredictionParameter.sMlModelFilePath := sModelJsonFilePath;
		fbMlSvr.stPredictionParameter.sMlSvrNetId := sMlSvrNetId;
		fbMlSvr.stPredictionParameter.eExecutionProvider := eExecutionProvider;
		IF fbMlSvr.Configure(nTimeout := nConfigureTimeout, nPriority := nPriority) THEN
			nErrorCode := fbMlSvr.nErrorCode;
			bError := fbMlSvr.bError OR (nErrorCode <> 0);
			bConfigured := fbMlSvr.bConfigured AND NOT(bError);
			bBusy := FALSE;
			IF bConfigured THEN
				nState := 20;
			ELSE
				nState := 90;
			END_IF
		END_IF

	20:
		bBusy := FALSE;
		bPredictionPending := FALSE;
		IF bEnable AND bConfigured AND NOT(bError) AND NOT(bReset) THEN
			FOR nSequenceIndex := 0 TO 32 DO
				stModelInput.in_input_tensor[0,nSequenceIndex,0] := fTheta + (INT_TO_REAL(nSequenceIndex) * fThetaStep);
				stModelInput.in_input_tensor[0,nSequenceIndex,1] := fThetaDot;
				stModelInput.in_input_tensor[0,nSequenceIndex,2] := fTorque;
				stModelInput.in_input_tensor[0,nSequenceIndex,3] := fTemperature;
			END_FOR
			bPredictionReady := FALSE;
			bPredictionPending := TRUE;
			nState := 30;
		END_IF

